(* CoDeSys 2.3.9.41 project: myLib.pro *)
(* Libraries: SysLibTime.lib 20.2.06 13:31:16, PID_Regulators.lib 28.12.06 17:47:54, Util.lib 18.5.10 15:14:28, STANDARD.LIB 4.10.05 11:14:46, IECSFC.LIB 13.4.06 15:51:28, ANALYZATION.LIB 5.10.99 09:05:06 *)

(* PLC configuration (modules and I/O channels)
Fast discrete inputs [I_SIMPLE_INPUT] node 0, in %IB0 out %QB0 {Filtrationtime = 10}
  DD1_DI0 AT %IX0.0 [BitInput] резерв
  DD1_DI1 AT %IX0.1 [BitInput] резерв
  DD1_DI2 AT %IX0.2 [BitInput] резерв
  DD1_DI3 AT %IX0.3 [BitInput] резерв
Discrete inputs [ID130] node 1, in %IB1 out %QB1 {Filtrationtime_GeneralINP = 10; Visibility = No; PinCount = 12}
  AT %IB1.0 [ByteInput] 8 discrete inputs
  AT %IB1.1 [ByteInput] 4 discrete inputs
Discrete outputs [ID131] node 2, in %IB2 out %QB2 {SafeValueByte = 0; SafeValueByteM = 0; Visibility = No; PinCount = 12}
  AT %QB2.0 [ByteOutput] 8 discrete outputs
  AT %QB2.1 [ByteOutput] 4 discrete outputs
Fast analog inputs [ID125] node 3, in %IB3 out %QB3 {Flt_Comm = 50Hz 2Por}
  DD1_AI0 AT %IR3.0 [FloatInputP] AI #1 - датчик температуры в помещении {AIN_TYPE = 4-20 mA; Peak_Filtr = 200; Flt_Ch = Off; TauRC = 10; MinFV = 0; MaxFV = 100}
  DD1_AI1 AT %IR3.1 [FloatInputP] AI #2 - расходомер FT01.01 (на входе, до отстойника) {AIN_TYPE = 4-20 mA; Peak_Filtr = 200; Flt_Ch = Off; TauRC = 10; MinFV = 0; MaxFV = 600}
  DD1_AI2 AT %IR3.2 [FloatInputP] AI #3 - расходомер FT01.02 (на выходе, после отстойника) {AIN_TYPE = 4-20 mA; Peak_Filtr = 200; Flt_Ch = Off; TauRC = 10; MinFV = 0; MaxFV = 600}
  DD1_AI3 AT %IR3.3 [FloatInputP] AI #4 - рН-метр QE01.01 (на входе, до отстойника) {AIN_TYPE = 4-20 mA; Peak_Filtr = 200; Flt_Ch = Off; TauRC = 10; MinFV = 0; MaxFV = 14}
  DD1_AI4 AT %IR3.4 [FloatInputP] AI #5 - рН-метр QE01.02 (на выходе, после отстойника) {AIN_TYPE = 4-20 mA; Peak_Filtr = 200; Flt_Ch = Off; TauRC = 10; MinFV = 0; MaxFV = 14}
  DD1_AI5 AT %IR3.5 [FloatInputP] AI #6 - сигнал от ФПК, давление на входе {AIN_TYPE = 4-20 mA; Peak_Filtr = 200; Flt_Ch = Off; TauRC = 10; MinFV = 0; MaxFV = 20000.0}
  DD1_AI6 AT %IR3.6 [FloatInputP] AI #7 - резерв {AIN_TYPE = 4-20 mA; Peak_Filtr = 200; Flt_Ch = Off; TauRC = 10; MinFV = 0; MaxFV = 20000.0}
  DD1_AI7 AT %IR3.7 [FloatInputP] AI #8 - обратная связь от ЧРП Н01.05 (частота, обороты, или ток) {AIN_TYPE = 4-20 mA; Peak_Filtr = 200; Flt_Ch = Off; TauRC = 10; MinFV = 0; MaxFV = 20000.0}
  AT %IW3.8 [WordInput] AI read time (10ms)
DD1_AO0 AT %QR4.0 [FloatOutputP] AO #1 - управление ЧРП Н01.05 (поддержание расхода по расходомеру FT01.02) {AOUT_TYPE = 4-20 mA; SafeValueREAL = 0.0}
DD1_AO1 AT %QR4.1 [FloatOutputP] AO #2 - управление ЧРП НД08.03/01 (подача флокулянта на входе, до отстойника, по FT01.01) {AOUT_TYPE = 4-20 mA; SafeValueREAL = 0.0}
DD1_AO2 AT %QR4.2 [FloatOutputP] AO #3 - управление ЧРП НД08.03/02 (подача флокулянта на входе, до отстойника, по FT01.01) {AOUT_TYPE = 4-20 mA; SafeValueREAL = 0.0}
DD1_AO3 AT %QR4.3 [FloatOutputP] AO #4 - управление НД05.02/01 (подача 10%NaCl из УПГ на входе, до отстойника, по FT01.01) {AOUT_TYPE = 4-20 mA; SafeValueREAL = 0.0}
Special input [ID103] node 5, in %IB5 out %QB5 {Filtrationtime = 1000; PinCount = 1; WatchDogPeriod = 400; PollPeriod = 3000; Visibility = No}
  AT %IX5.0 [BitInput] Special input
Special output [ID104] node 6, in %IB6 out %QB6 {Visibility = No; PinCount = 1}
  AT %QX6.0 [BitOutput] Special output
ModBus (Master) [MODBUS_MASTER_ID450] node 7, in %IB7 out %QB7 {Visibility = No}
  AT %QD7.0 [DWordOutput] Last address
  AT %QW7.1 [WordOutput] Last error
  RS-485-1 [COM1_USART] node 0, in %IB7.0 out %QB7.0 {CommunicationSpeed = 57600; Parity = NO PARITY CHECK; BitLength = 8 bits; StopLength = One stop bit; InterfaceType = RS485; FrameOriented = RTU; Timeout = 0; Visibility = No}
  Universal Modbus device [ID2000] node 1, in %IB7.1 out %QB7.1 {ModuleIP = 10:0:0:102; ServiceTimeout = 20; TCPport = 502; NetMode = Serial; ModuleSlaveAddress = 2; RequestType = Both; PeriodOfService = 100; Visibility = No; RepeatCounter = 0; ByteSequence = Trace_mode}
    AT %QB7.1.0 [ComChannel] Command (0xff - Start)
DD2_DO AT %QD7.1.0.0 [DWordOutput] регистр 0, команда 0х0f
Universal Modbus device [ID2000] node 2, in %IB7.2 out %QB7.2 {ModuleIP = 10:0:0:103; ServiceTimeout = 20; TCPport = 502; NetMode = Serial; ModuleSlaveAddress = 3; RequestType = Both; PeriodOfService = 100; Visibility = No; RepeatCounter = 0; ByteSequence = Trace_mode}
  AT %QB7.2.0 [ComChannel] Command (0xff - Start)
DD3_DO AT %QD7.2.0.0 [DWordOutput]
Universal Modbus device [ID2000] node 3, in %IB7.3 out %QB7.3 {ModuleIP = 10:0:0:104; ServiceTimeout = 20; TCPport = 502; NetMode = Serial; ModuleSlaveAddress = 4; RequestType = Both; PeriodOfService = 100; Visibility = No; RepeatCounter = 0; ByteSequence = Trace_mode}
  AT %QB7.3.0 [ComChannel] Command (0xff - Start)
  32bit output module [ID2006] node 0, in %IB7.3.0 out %QB7.3.0 {ModbusAddress = 0; Command_write_regs = Force multiple coils (0x0f); Visibility = No}
    DD4_DO AT %QD7.3.0.0 [DWordOutput]
Universal Modbus device [ID2000] node 4, in %IB7.4 out %QB7.4 {ModuleIP = 10:0:0:105; ServiceTimeout = 20; TCPport = 502; NetMode = Serial; ModuleSlaveAddress = 5; RequestType = Both; PeriodOfService = 100; Visibility = No; RepeatCounter = 0; ByteSequence = Trace_mode}
  AT %QB7.4.0 [ComChannel] Command (0xff - Start)
DD5_DI AT %ID7.4.0.0 [DWordInput]
Universal Modbus device [ID2000] node 5, in %IB7.5 out %QB7.5 {ModuleIP = 10:0:0:106; ServiceTimeout = 20; TCPport = 502; NetMode = Serial; ModuleSlaveAddress = 6; RequestType = Both; PeriodOfService = 100; Visibility = No; RepeatCounter = 0; ByteSequence = Trace_mode}
  AT %QB7.5.0 [ComChannel] Command (0xff - Start)
DD6_DI AT %ID7.5.0.0 [DWordInput]
Universal Modbus device [ID2000] node 6, in %IB7.6 out %QB7.6 {ModuleIP = 10:0:0:107; ServiceTimeout = 20; TCPport = 502; NetMode = Serial; ModuleSlaveAddress = 7; RequestType = Both; PeriodOfService = 100; Visibility = No; RepeatCounter = 0; ByteSequence = Trace_mode}
  AT %QB7.6.0 [ComChannel] Command (0xff - Start)
DD7_DI AT %ID7.6.0.0 [DWordInput]
Universal Modbus device [ID2000] node 7, in %IB7.7 out %QB7.7 {ModuleIP = 10:0:0:108; ServiceTimeout = 20; TCPport = 502; NetMode = Serial; ModuleSlaveAddress = 8; RequestType = Both; PeriodOfService = 100; Visibility = No; RepeatCounter = 0; ByteSequence = Trace_mode}
  AT %QB7.7.0 [ComChannel] Command (0xff - Start)
DD8_DI AT %ID7.7.0.0 [DWordInput]
Universal Modbus device [ID2000] node 8, in %IB7.8 out %QB7.8 {ModuleIP = 10:0:0:109; ServiceTimeout = 20; TCPport = 502; NetMode = Serial; ModuleSlaveAddress = 9; RequestType = Both; PeriodOfService = 100; Visibility = No; RepeatCounter = 0; ByteSequence = Trace_mode}
  AT %QB7.8.0 [ComChannel] Command (0xff - Start)
DD9_DI AT %ID7.8.0.0 [DWordInput]
AT %QB7.9.0 [ComChannel] Command (0xff - Start)
DD10_AO0 AT %QW7.9.0.0 [WordOutput] управление 4...20мА НД05.02/01
DD10_AO1 AT %QW7.9.1.0 [WordOutput]
DD10_AO2 AT %QW7.9.2.0 [WordOutput]
DD10_AO3 AT %QW7.9.3.0 [WordOutput]
DD10_AO4 AT %QW7.9.4.0 [WordOutput]
DD10_AO5 AT %QW7.9.5.0 [WordOutput]
DD10_AO6 AT %QW7.9.6.0 [WordOutput]
DD10_AO7 AT %QW7.9.7.0 [WordOutput]
*)

(* Global variable list: Global_Variables *)
VAR_GLOBAL
	wordMaxValue: WORD := 65535;		(*max value of WORD.*)
END_VAR

(* POU PLC_PRG, CFC *)
PROGRAM PLC_PRG
VAR
	temperatureLimits: LIMITALARM;		(*блок контроля границ допустимой температуры в помещении*)
	alarmHighTemperature: BOOL;		(*температура выше заданного диапазона*)
	alarmLowTemperature: BOOL;		(*температура ниже заданного диапазона*)
	temperatureValue: REAL;		(*значение температуры в помещении*)
	DD1_AI0_temperature: DECODE_FLOAT;		(*блок контроля состояния аналогового входа ПЛК для датчика температуры в помещении*)
	DD1_AI1_flow: DECODE_FLOAT;		(*блок контроля состояния аналогового входа ПЛК для расходомера FT01.01*)

	ND0502dosing: DosingPumpProportional;		(*Блок управления дозированием насосов НД05.02/01 и НД05.02/02.
			Пропорционально расходу по FT01.01*)
	ND0502regime: choosePumpRegime;		(*Блок выбора режима включения НД05.02/01 и НД05.02/02.*)
	ND0502manager: TwoPumpManager;		(*Блок управления включением дозирующих насосов
			НД05.02/01 и НД05.02/02.*)

	ND0602dosing: DosingPumpProportional;		(*Блок управления дозированием насосов НД06.02/01 и НД06.02/02.
			Пропорционально расходу по FT01.02.*)
	ND0602regime: choosePumpRegime;		(*Блок выбора режима включения НД06.02/01 и НД06.02/02.*)
	ND0602manager: TwoPumpManager;		(*Блок управления включением дозирующих насосов
			НД06.02/01 и НД06.02/02.*)

	ND0603dosing: DosingPumpProportional;		(*Блок управления дозированием насосов НД06.03/01 и НД06.03/02.
						Пропорционально расходу по FT01.01*)
	ND0603regime: choosePumpRegime;		(*Блок выбора режима включения НД06.03/01 и НД06.03/02.*)
	ND0603manager: TwoPumpManager;		(*Блок управления включением дозирующих насосов
						НД06.03/01 и НД06.03/02.*)

	ND0703pidReg: PID;		(*Блок автоматического поддержания заданного значения рН стоков подачей щелочи через НД07.03
								по показаниям QE01.01.*)
	ND0703regime: choosePumpRegime;		(*Блок выбора режима включения НД07.03/01 и НД07.03/02.*)
	ND0703manager: TwoPumpManager;		(*Блок управления включением дозирующих насосов
									НД07.03/01 и НД07.03/02*)

	ND0803dosing: DosingPumpProportional;		(*Блок управления дозированием насосов НД08.03*)
	ND0803regime: choosePumpRegime;		(*Блок выбора режима включения насосов НД08.03.*)
	ND0803manager: TwoPumpManager;		(*Блок управления включением дозирующих насосов НД08.03.*)

	ND0804linearTransformator: LIN_TRAFO;		(*Блок преобразования сигнала на управление от 0 до 100% в 4...20мА*)

	DD1_AI1_FT0101: DECODE_FLOAT;		(*Блок контроля аналогового входа DD1_AI1 (расходомер FT01.01)*)
	DD1_AI2_FT0102: DECODE_FLOAT;		(*блок контроля состояния аналогового входа ПЛК для расходомера FT01.02*)
	DD1_AI3_QE0101: DECODE_FLOAT;		(*блок контроля состояния аналогового входа ПЛК для рН-метра QE01.01*)
	DD1_AI4_QE0102: DECODE_FLOAT;		(*блок контроля состояния аналогового входа ПЛК для рН-метра QE01.02*)

	DD1_AI1_FT0101value: REAL;		(*Показания расходомера FT01.01 после блока контроля аналогового входа ПЛК.*)
	DD1_AI2_FT0102value: REAL;		(*Показания расходомера FT01.02 после блока контроля аналогового входа ПЛК.*)
	DD1_AI3_QE0101value: REAL;		(*Показания рН-метра QE01.01 после блока контроля аналогового входа ПЛК.*)
	DD1_AI4_QE0102value: REAL;		(*Показания рН-метра QE01.02 после блока контроля аналогового входа ПЛК*)

	N0105manager: TwoPumpManager;		(*Блок управления включением насосов Н01.05*)
	N0105regime: choosePumpRegime;		(*Блок выбора режима включения Н05.01*)
	N0105pidReg: PID;		(*Блок автоматического поддержания заданного значения расхода по показаниям FT01.02*)
	N0105regByC: RS;		(*Триггер выбора режима по количеству включений.*)
	N0105regByWT: RS;		(*Триггер выбора режима по наработке.*)
	N0105managerKM1off: BOOL;		(*Переменная управления состоянием контактора питания ЧРП (КМ1).*)
	N0105rsTrigKM1: RS;		(*Триггер управления состоянием контактора КМ1. Постоянно включен.
			Выключается если N0105managerKM1off=true.*)
	N0105timerKM1off: TOF;		(*Таймер отключения КМ1. Срабатывает по импульсу на входе.
			Выключается через заданное в N0105switchKM1Delay время.*)
	N0105switchKM1Delay: TIME := T#20S;		(*Время отключения питания ЧРП Н01.05.
			По умолчанию = 20 сек.*)
	N010501rTrig: R_TRIG;		(*Детектор перенего фронта сигнала выбора режима Н01.05/01 = главный.*)
	N010501fTrig: F_TRIG;		(*Детектор спада сигнала выбора режима Н01.05/01 = главный.*)
	N0105trigKM2on: RS;		(*Триггер включения КМ2.*)
	N0105switchKM2Delay: TON;		(*Таймер задержки включения КМ2.*)
	N0105switchKM23Delay: TIME := T#15s;		(*Время задержки включения КМ2 и КМ3 при переключении.
			По умолчанию 15 сек.*)
	N010502rTrig: R_TRIG;		(*Детектор перенего фронта сигнала выбора режима Н01.05/02 = главный.*)
	N010502fTrig: F_TRIG;		(*Детектор спада сигнала выбора режима Н01.05/02 = главный.*)
	N0105trigKM3on: RS;		(*Триггер включения КМ3.*)
	N0105switchKM3Delay: TON;		(*Таймер задержки включения КМ3.*)

	rTrigStartInitializer: R_TRIG;		(*Детектор переднего фронта,
			инициализирует булевы переменные при старте программы.*)
	startInitializer: BOOL;		(*Инициализирует булевы переменные при старте программы.*)

	N0105sttartTrig: RS;		(*Триггер запуска насосов Н01.05 по датчикам уровня.*)

	N010501alarm: BOOL;		(*Авария насоса Н01.05/01*)
	N010502alarm: BOOL;		(*Авария насоса Н01.05/02*)
	N010501toStart: BOOL;		(*Промежуточный сигнал о необходимости запуска Н01.05/01.*)
	N010502toStart: BOOL;		(*Промежуточный сигнал о необходимости запуска Н01.05/02.*)
	N0105minFlow: REAL := 10;		(*Минимальное значение расхода для подачи сигнала на начало дозирования.
			По умолчанию, если ничего не подключено ко входу, равно 10 кубометров в час.*)
	N0105f_trigStop: F_TRIG;		(*Детектор останова насоса кнопкой со щита (спад сигнала включенного реле).*)
	N010501alarmTrig: RS;		(*Триггер аварии насоса Н01.05/01.*)
	N010502alarmTrig: RS;		(*Триггер аварии насоса Н01.05/02.*)



	tempN0105switchKM1off: BOOL;		(*temporary variable to switch off KM1 when pumps change.*)
	tempN010501Trig: RS;		(*temporary trigger to catch N010501 start impuls.*)
	tempN010502Trig: RS;		(*temporary trigger to catch N01.05/02 start impuls*)
	tempN0105rTrigKM1off: R_TRIG;		(*temporary rising front detector to switch off KM1 = drive power supply.*)
	tempN010501rTrig: R_TRIG;		(*temporary rising signal to start N010501 detector*)
	tempN010502rTrig: R_TRIG;		(*temporary rising signal to start N010502 detector*)
	tempN0105RMswitchDelay: BOOL;		(*Init temporaty delay to switch KM2 or KM3.*)
	tempN0105delayOUT: BOOL;		(*temporari signal that delay to switch is over.*)
	tempN0105switchKM2offDelay: TOF;		(*temporary delay to switch off KM2*)
	tempN0105switchKM3offDelay: TOF;		(*temporary delay to switch off KM3*)
	tempN0105switchKMoffDelay: TIME := T#3s;		(*temporary switch off RM delay.*)
	tempN0105ready: BOOL;		(*Temporary variable shows that system is ready to start pump.*)
	tempN0105readyToStart: TON;		(*Temporary ready to start delay timer.*)
	tempN0105readyToStartDelay: TIME := T#5s;		(*temporary delay to show signal that system is ready to start.
			Init value = 5sec.*)
	tempTwoPumpOneDriveManager: TwoPumpOneDriveManager;		(*test*)
	temp1: BOOL;
	temp2: BOOL;
	temp3: BOOL;
	temp4: BOOL;
	temp5: BOOL;
	temp6: BOOL;
	temp7: BOOL;
	temp8: BOOL;
	temp9: BOOL;
	temp10: BOOL;
	temp11: BOOL;
	temp12: WORD;
	temp13: WORD;
	temp14: TIME;
	temp15: TIME;
	temp16: BOOL;
	temp17: BOOL;
	temp18: BOOL;
	temp19: BOOL;
END_VAR
VAR_INPUT
	alarmReset: BOOL;		(*Сброс аварий.*)

	ND0502resetCountP1: BOOL;		(*Сбросить счетчик количества включений НД05.02/01.*)
	ND0502resetCountP2: BOOL;		(*Сбросить счетчик количества включений НД05.02/02.*)
	ND0502resetWorkTimeP1: BOOL;		(*Сбросить счетчик наработки НД05.02/01.*)
	ND0502resetWorkTimeP2: BOOL;		(*Сбросить счетчик наработки НД05.02/02.*)

	ND0602resetCountP1: BOOL;		(*Сбросить счетчик количества включений НД06.02/01.*)
	ND0602resetCountP2: BOOL;		(*Сбросить счетчик количества включений НД06.02/02.*)
	ND0602resetWorkTimeP1: BOOL;		(*Сбросить счетчик количества наработки НД06.02/01.*)
	ND0602resetWorkTimeP2: BOOL;		(*Сбросить счетчик количества наработки НД06.02/02.*)

	ND0603resetCountP1: BOOL;		(*Сбросить счетчик количества включений НД06.03/01.*)
	ND0603resetCountP2: BOOL;		(*Сбросить счетчик количества включений НД06.03/02.*)
	ND0603resetWorkTimeP1: BOOL;		(*Сбросить счетчик времени наработки НД06.03/01.*)
	ND0603resetWorkTimeP2: BOOL;		(*Сбросить счетчик времени наработки НД06.03/02.*)

	ND0703resetCountP1: BOOL;		(*Сбросить счетчик количества включений НД07.03/01.*)
	ND0703resetCountP2: BOOL;		(*Сбросить счетчик количества включений НД07.03/02.*)
	ND0703resetWorkTimeP1: BOOL;		(*Сбросить счетчик наработки НД07.03/01.*)
	ND0703resetWorkTimeP2: BOOL;		(*Сбросить счетчик наработки НД07.03/02.*)
	ND0703YoutManual: REAL;		(*Задание значения выходу Y в ручном режиме (4...20мА).*)
	ND0703YmanAuto: BOOL;		(*Выбор управления выходом Y в ручном или автоматическом режиме.*)

	ND0803resetCountP1: BOOL;		(*Сброс счетчика количества включений НД08.03/01.*)
	ND0803resetCountP2: BOOL;		(*Сброс счетчика количества включений НД08.03/02.*)
	ND0803resetWorkTimeP1: BOOL;		(*Сброс счетчика наработки НД08.03/01.*)
	ND0803resetWorkTimeP2: BOOL;		(*Сброс счетчика наработки НД08.03/02.*)

	N0105YoutManual: REAL;		(*Задание значения выходу Y в ручном режиме (4...20мА).*)
	N0105YmanAuto: BOOL;		(*Выбор управления выходом Y в ручном или автоматическом режиме.*)

END_VAR
VAR_OUTPUT
	ND0502dosingError: BOOL;		(*Ошибка дозирования НД05.02.
			Проверить заданные уставки.*)
	ND0502statRegimeP1M: BOOL;		(*статус: режим НД05.02 - насос 1 = главный.*)
	ND0502statRegimeP2M: BOOL;		(*статус: режим НД05.02 - насос 2 = главный*)
	ND0502statRegimeByC: BOOL;		(*статус: режим НД05.02 - по количеству включений*)
	ND0502statRegimeByWT: BOOL;		(*статус: режим НД05.02 - по наработке*)

	ND0602dosingError: BOOL;		(*Ошибка дозирования НД06.02/01-02.
						Проверить заданные уставки.*)
	ND0602statRegimeP1M: BOOL;		(*статус: режим НД0602 - насос 1 = главный.*)
	ND0602statRegimeP2M: BOOL;		(*статус: режим НД06.02 - насос 2 = главный.*)
	ND0602statRegimeByC: BOOL;		(*статус: режим НД06.02 - по количеству включений.*)
	ND0602statRegimeByWT: BOOL;		(*статус: режим НД06.02 - по наработке.*)

	ND0603dosingError: BOOL;		(*Ошибка дозирования НД06.03.
						Проверить заданные уставки.*)
	ND0603statRegimeP1M: BOOL;		(*статус: режим НД0603 - насос 1 = главный.*)
	ND0603statRegimeP2M: BOOL;		(*статус: режим НД0603 - насос 2 = главный.*)
	ND0603statRegimeByC: BOOL;		(*статус: режим НД06.03 - по количеству включений.*)
	ND0603statRegimeByWT: BOOL;		(*статус: режим НД06.03 - по наработке.*)

	ND0703statRegimeP1M: BOOL;		(*статус: режим НД0703 - насос 1 = главный.*)
	ND0703statRegimeP2M: BOOL;		(*статус: режим НД0703 - насос 2 = главный.*)
	ND0703statRegimeByC: BOOL;		(*статус: режим НД07.03 - по количеству включений.*)
	ND0703statRegimeByWT: BOOL;		(*статус: режим НД07.03 - по наработке.*)

	ND0803dosingError: BOOL;		(*Ошибка блока дозирования НД08.03.*)
	ND0803statRegimeP1M: BOOL;		(*статус: режим НД08.03 - насос 1 = главный*)
	ND0803statRegimeP2M: BOOL;		(*статус: режим НД08.03 - насос 2 = главный*)
	ND0803statRegimeByC: BOOL;		(*статус: режим НД08.03 - по количеству включений*)
	ND0803statRegimeByWT: BOOL;		(*статус: режим НД08.03 - по наработке.*)

	ND0804dosingError: BOOL;		(*Ошибка дозирования НД08.04. Проверь уставки.*)

	DD1_AI0_error: BOOL;		(*авария входа AI1 (возможно, обрыв)*)
	DD1_AI1_error: BOOL;		(*авария входа AI2 (возможно, обрыв)*)
	DD1_AI2_error: BOOL;		(*авария входа AI3 (возможно, обрыв)*)
	DD1_AI3_error: BOOL;		(*авария входа AI4 (возможно, обрыв)*)
	DD1_AI4_error: BOOL;		(*авария входа AI5 (возможно, обрыв)*)

	N0105statRegimeP1M: BOOL;		(*статус: режим Н01.05/01 = главный.*)
	N0105statRegimeP2M: BOOL;		(*статус: режим Н01.05/02 = главный.*)
	N0105statRegimeByC: BOOL;		(*статус: режим Н01.05 = по количеству включений.*)
	N0105statRegimeByWT: BOOL;		(*статус: режим Н01.05 = по наработке.*)

END_VAR
VAR RETAIN
	maxTemperature: BYTE;		(*Температура, выше которой будет подан сигнал ВЫСОКАЯ ТЕМПЕРАТУРА*)
	minTemperature: BYTE;		(*температура, ниже которой будет подан сигнал НИЗКАЯ ТЕМПЕРАТУРА*)

END_VAR
VAR_INPUT RETAIN
	ND0502setMaxDosVal: REAL;		(*Указать максимальную производительность НД05.02.*)
	ND0502setKoefProp: REAL;		(*Задать количество реагента в мл на один кубометр стоков.*)
	ND0502regimeP1M: BOOL := 1;		(*Выбор режима включения доз.насосов НД05.02: первый насос - главный.
			Выбрано по умолчанию до выбора пользователя.*)
	ND0502regimeP2M: BOOL;		(*Выбор режима включения доз.насосов НД05.02:
			второй насос - главный.*)
	ND0502regimeByWT: BOOL;		(*Выбор режима включения доз.насосов НД05.02:
			по наработке.*)
	ND0502regimeByC: BOOL;		(*Выбор режима включения доз.насосов НД05.02:
			по количеству включений.*)

	ND0602setMaxDosVal: REAL;		(*Указать максимальную производительность НД06.02.*)
	ND0602setKoefProp: REAL;		(*Задать количество реагента в мл на один кубометр стоков.*)
	ND0602regimeP1M: BOOL := 1;		(*Выбор режима включения доз.насосов НД06.02: первый насос - главный.
			Выбрано по умолчанию до выбора пользователя.*)
	ND0602regimeP2M: BOOL;		(*Выбор режима включения доз.насосов НД06.02: второй насос - главный.
			*)
	ND0602regimeByWT: BOOL;		(*Выбор режима включения доз.насосов НД06.02:
			по наработке.*)
	ND0602regimeByC: BOOL;		(*Выбор режима включения доз.насосов НД06.02:
			по количеству включений.*)

	ND0603setMaxDosVal: REAL;		(*Указать максимальную производительность НД06.03.*)
	ND0603setKoefProp: REAL;		(*Задать количество реагента в мл на один кубометр стоков.*)
	ND0603regimeP1M: BOOL := 1;		(*Выбор режима включения доз.насосов НД06.03: первый насос - главный.
			Выбрано по умолчанию до выбора пользователя.*)
	ND0603regimeP2M: BOOL;		(*Выбор режима включения доз.насосов НД06.03: второй насос - главный.*)
	ND0603regimeByWT: BOOL;		(*Выбор режима включения доз.насосов НД06.03:
			по наработке.*)
	ND0603regimeByC: BOOL;		(*Выбор режима включения доз.насосов НД06.03:
			по количеству включений.*)

	ND0703pHsetValue: REAL := 7.5;		(*Задание рН для поддержания подачей щелочи НД07.03 и контроля по QE01.01.*)
	ND0703regimeP1M: BOOL := 1;		(*Выбор режима включения доз.насосов НД07.03: первый насос - главный.
						Выбрано по умолчанию до выбора пользователя.*)
	ND0703regimeP2M: BOOL;		(*Выбор режима включения доз.насосов НД07.03: второй насос - главный*)
	ND0703regimeByWT: BOOL;		(*Выбор режима включения доз.насосов НД07.03: по наработке.*)
	ND0703regimeByC: BOOL;		(*Выбор режима включения доз.насосов НД07.03: по количеству включений.*)
	ND0703koeffI: REAL := 10;		(*Коэффициент интегральной части ПИД. По умолчанию = 10.*)
	ND0703koeffD: REAL := 1;		(*Коэффициент дифференциальной части ПИД. По умолчанию = 1.*)
	ND0703koeffP: REAL := 1;		(*Коэффициент пропорциональной части ПИД. По умолчанию = 1.*)

	ND0803setMaxDosVal: REAL;		(*Указать максимальную производительность НД08.03*)
	ND0803setKoefProp: REAL;		(*Задать количество реагента в мл на один кубометр стоков.*)
	ND0803regimeP1M: BOOL := 1;		(*Выбор режима включения доз.насосов НД08.03: первый насос - главный.
									Выбрано по умолчанию до выбора пользователя.*)
	ND0803regimeP2M: BOOL;		(*Выбор режима включения доз.насосов НД08.03: второй насос - главный.*)
	ND0803regimeByWT: BOOL;		(*Выбор режима включения доз.насосов НД08.03: по наработке.*)
	ND0803regimeByC: BOOL;		(*Выбор режима включения доз.насосов НД08.03: по количеству включений.*)

	ND0804doseValue: BYTE;		(*Задание на дозирование НД0804 в процентах от максимальной производительности (0-100).*)

	N0105regimeByC: BOOL;		(*Выбор режима запуска Н01.05: по количеству включений.
			*)
	N0105regimeByWT: BOOL;		(*Выбор режима запуска Н01.05: по наработке.*)
	N0105flowSetValue: REAL := 72;		(*Задание расхода для поддержания ЧРП Н01.05 по расходомеру FT01.02.
			По умолчанию = 72 кубометра в час.*)
	N0105koeffP: REAL := 1;		(*Коэффициент пропорциональной части ПИД. По умолчанию = 1.*)
	N0105koeffI: REAL := 10;		(*Коэффициент интегральной части ПИД. По умолчанию = 10.*)
	N0105koeffD: REAL := 1;		(*Коэффициент дифференциальной части ПИД. По умолчанию = 1.*)

END_VAR
VAR_OUTPUT RETAIN
	ND0502counterP1: WORD;		(*Счетчик количества включений НД05.02/01.*)
	ND0502counterP2: WORD;		(*Счетчик количества включений НД05.02/02.*)
	ND0502workTimeP1: TIME;		(*Счетчик времени наработки НД05.02/01.*)
	ND0502workTimeP2: TIME;		(*Счетчик времени наработки НД05.02/02.*)

	ND0602counterP1: WORD;		(*Счетчик количества включений НД06.02/01.*)
	ND0602counterP2: WORD;		(*Счетчик количества включений НД06.02/02.*)
	ND0602workTimeP1: TIME;		(*Счетчик времени наработки НД06.02/01.*)
	ND0602workTimeP2: TIME;		(*Счетчик времени наработки НД06.02/02.*)

	ND0603counterP1: WORD;		(*Счетчик количества включений НД06.03/01.*)
	ND0603counterP2: WORD;		(*Счетчик количества включений НД06.03/02.*)
	ND0603workTimeP1: TIME;		(*Счетчик времени наработки НД06.03/01.*)
	ND0603workTimeP2: TIME;		(*Счетчик времени наработки НД06.03/02.*)

	ND0703counterP1: WORD;		(*Счетчик количества включений НД07.03/01.*)
	ND0703counterP2: WORD;		(*Счетчик количества включений НД07.03/02.*)
	ND0703workTimeP1: TIME;		(*Счетчик времени наработки НД07.03/01.*)
	ND0703workTimeP2: TIME;		(*Счетчик времени наработки НД07.03/02.*)

	ND0803counterP1: WORD;		(*Счетчик количества включений НД08.03/01.*)
	ND0803counterP2: WORD;		(*Счетчик количества включений НД08.03/02.*)
	ND0803workTimeP1: TIME;		(*Счетчик времени наработки НД08.03/01.*)
	ND0803workTimeP2: TIME;		(*Счетчик времени наработки НД08.03/02.*)

	N0105counterP1: WORD;		(*Счетчик количества включений Н01.05/01.*)
	N0105counterP2: WORD;		(*Счетчик количества включений Н01.05/02.*)
	N0105workTimeP1: TIME;		(*Счетчик времени наработки Н01.05/01.*)
	N0105workTimeP2: TIME;		(*Счетчик времени наработки Н01.05/02.*)
END_VAR
VAR (* helpers for the ST form of the networks *)
	_t977 : WORD;
	_t899 : WORD;
	_t831 : REAL;
	_t801 : WORD;
	_t1027 : WORD;
	_t1033 : WORD;
	_t1355 : REAL;
	_t1361 : REAL;
	_t1183 : WORD;
	_t1189 : WORD;
	_t1404 : BOOL;
	_t1403 : BOOL;
END_VAR
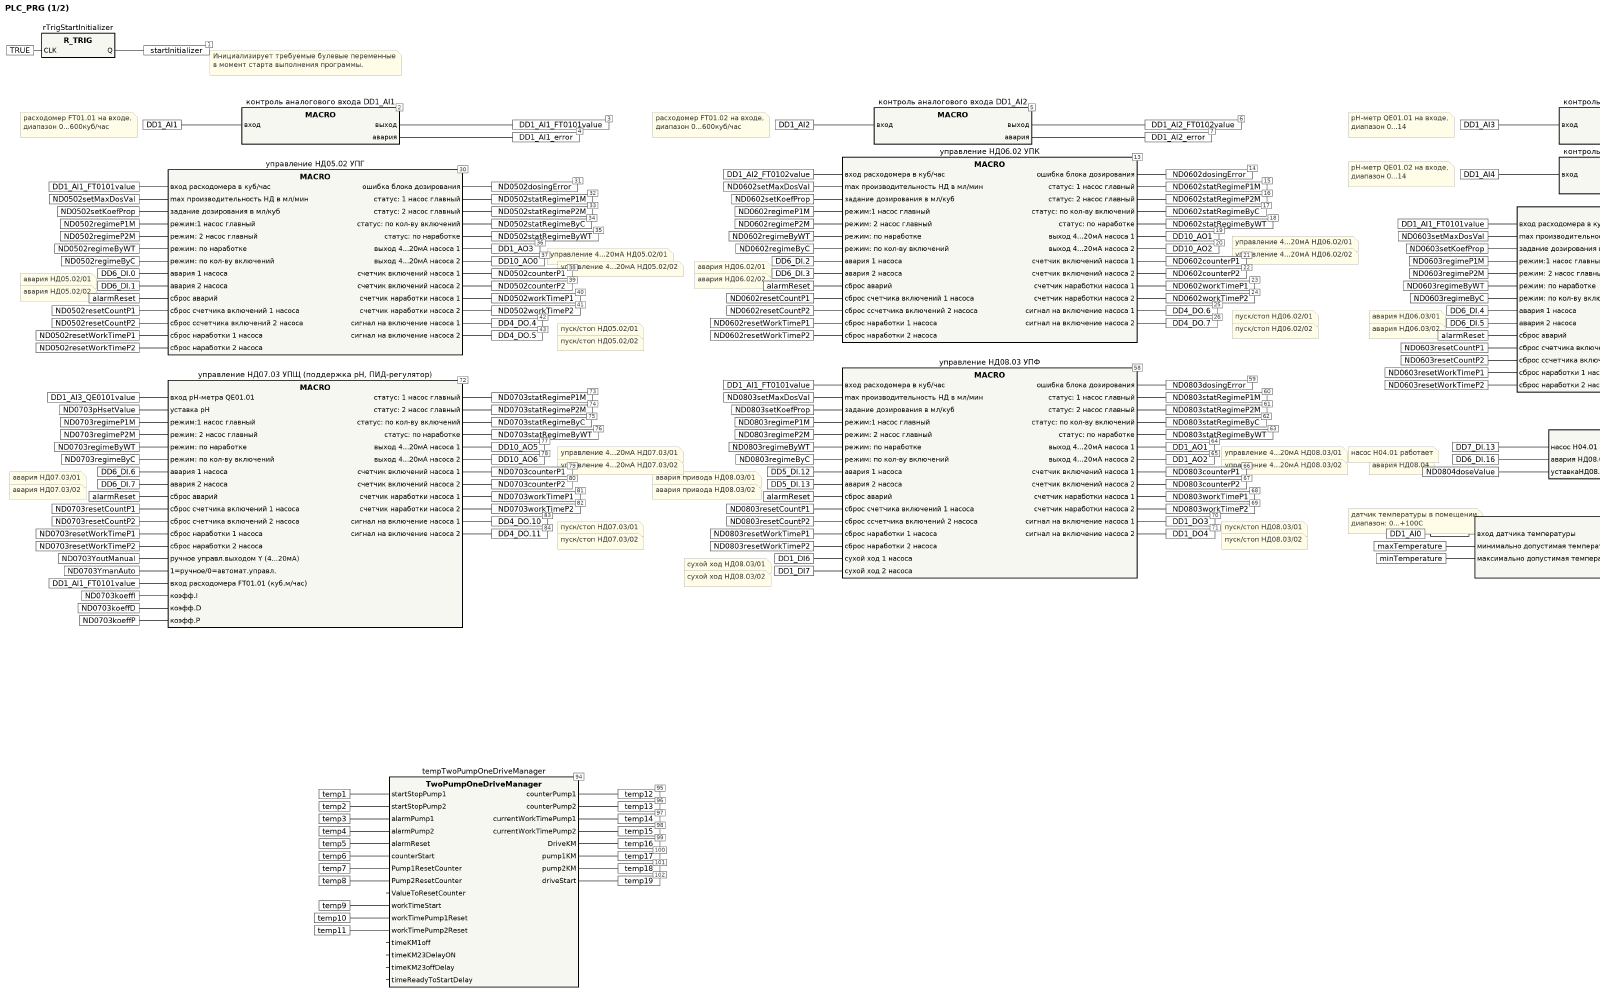
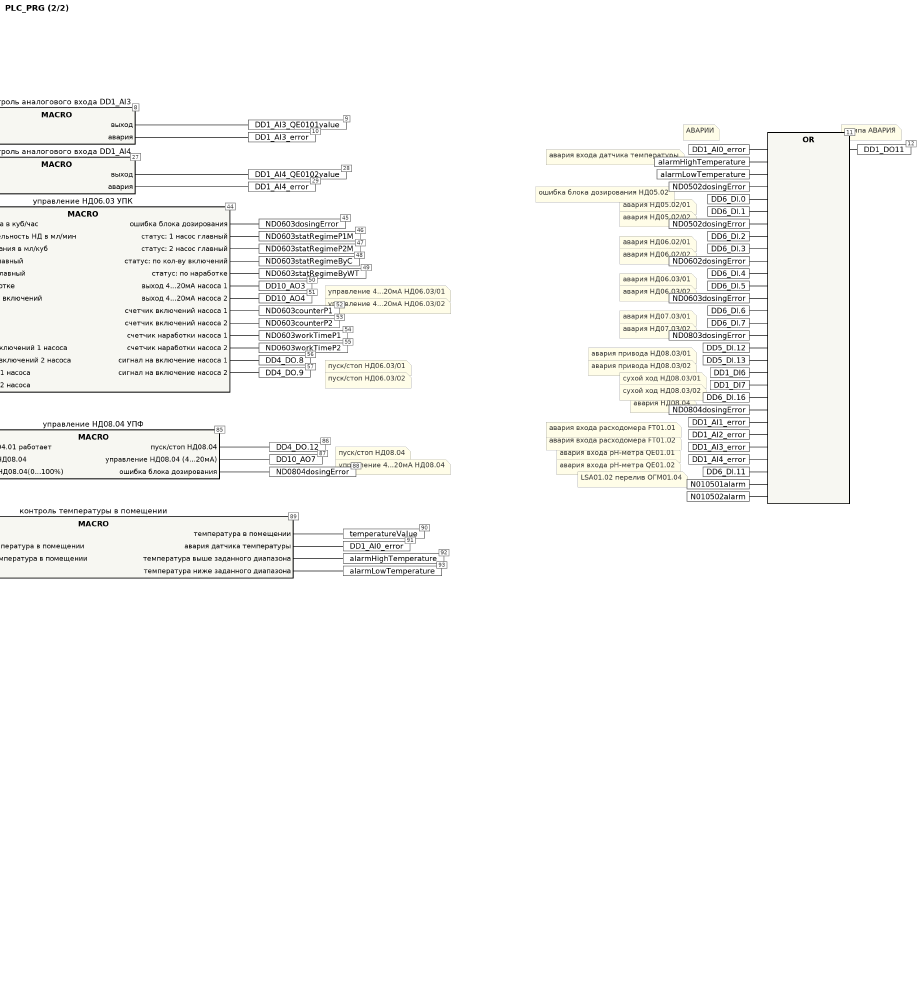
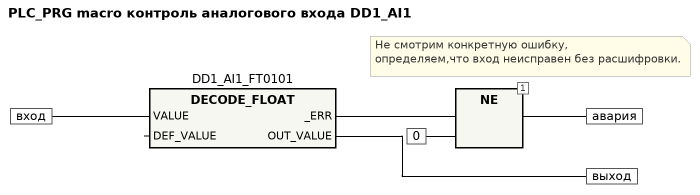
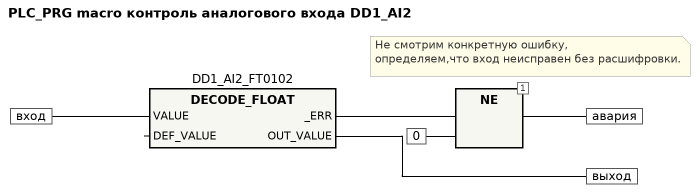
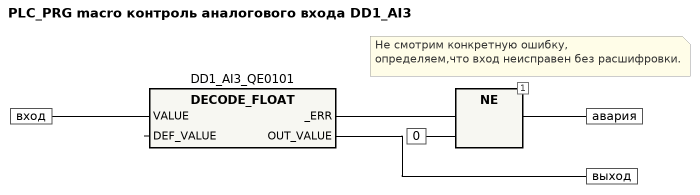
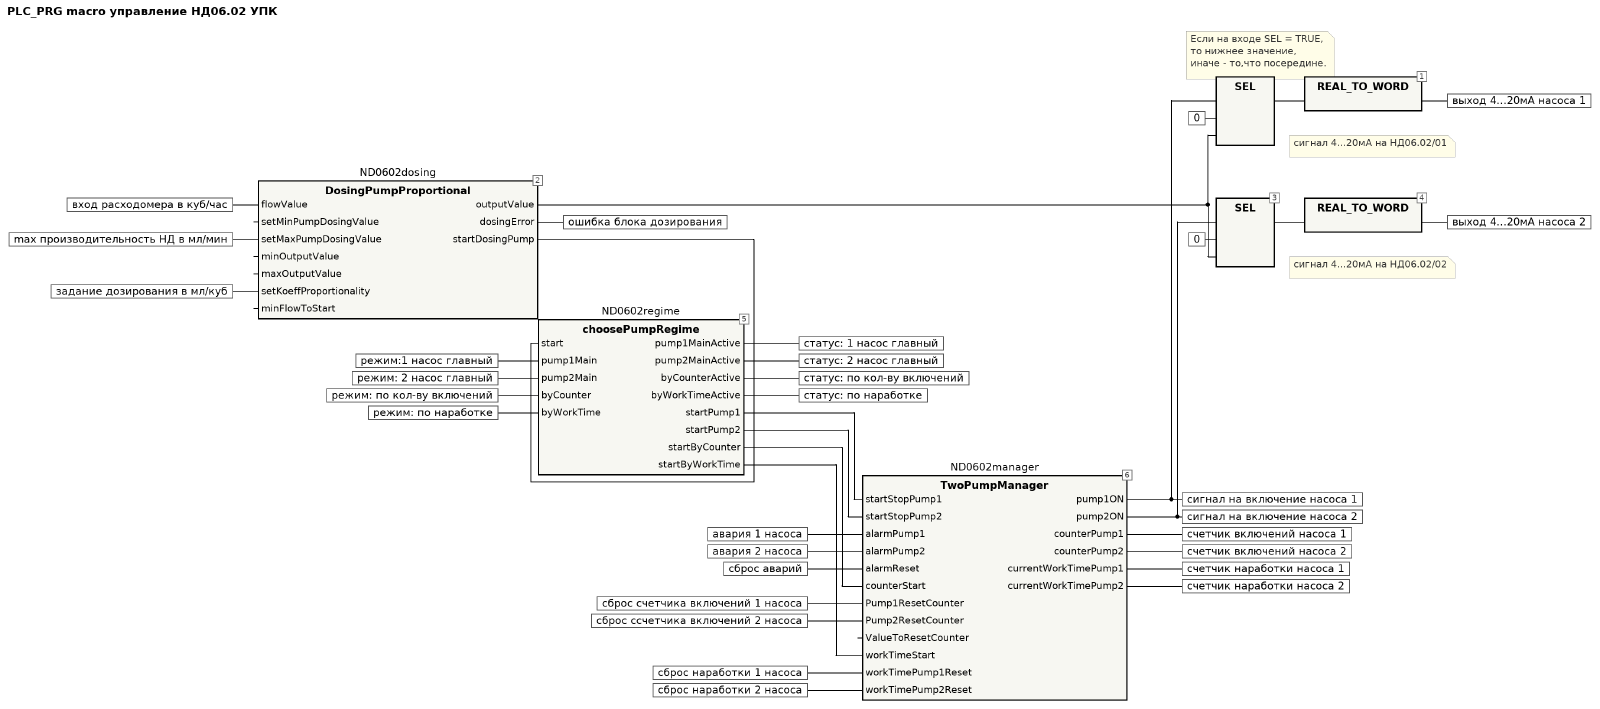
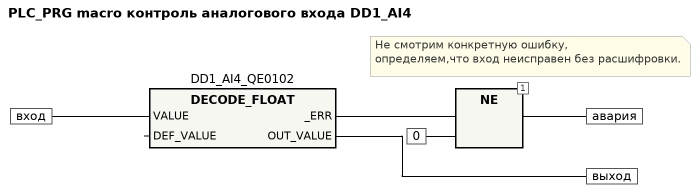
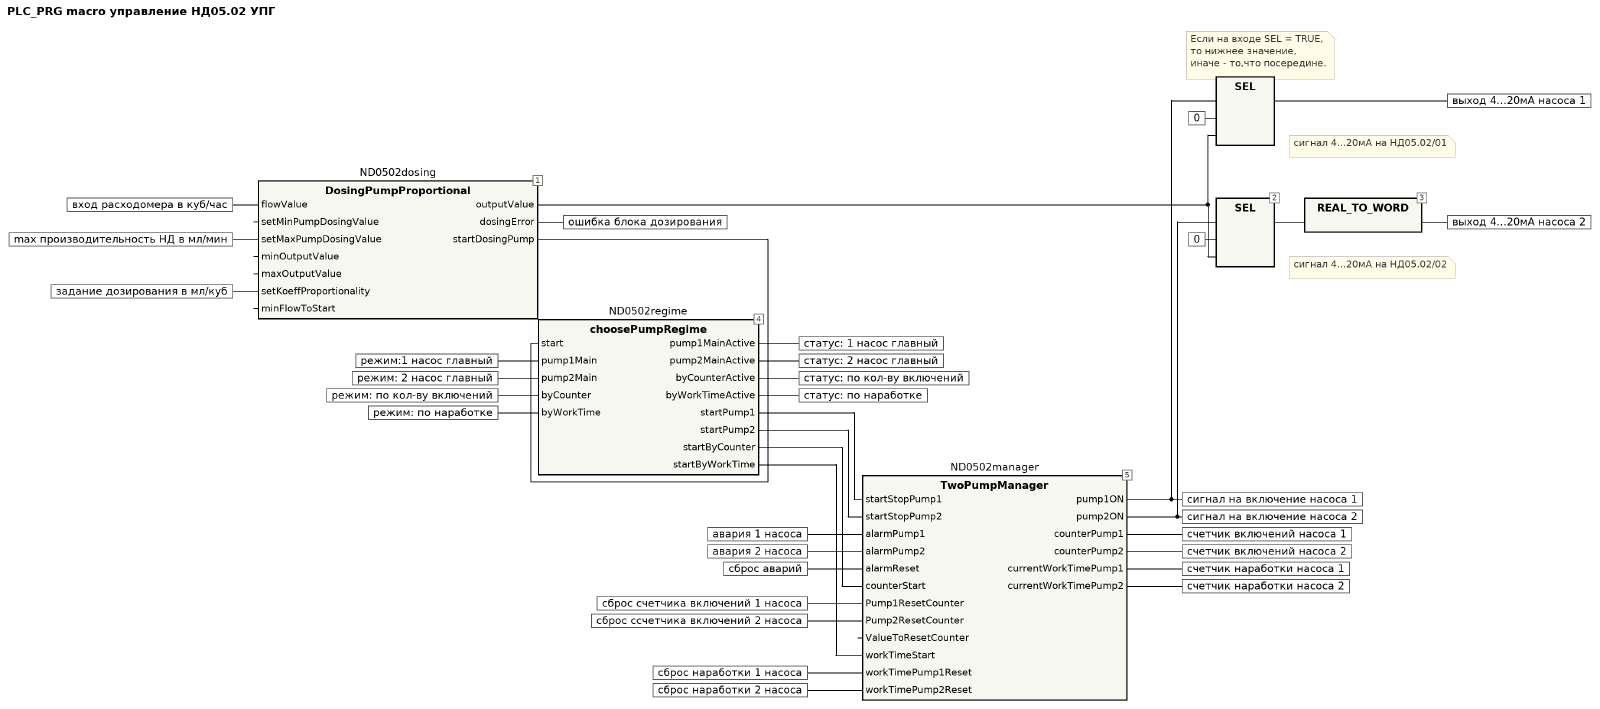
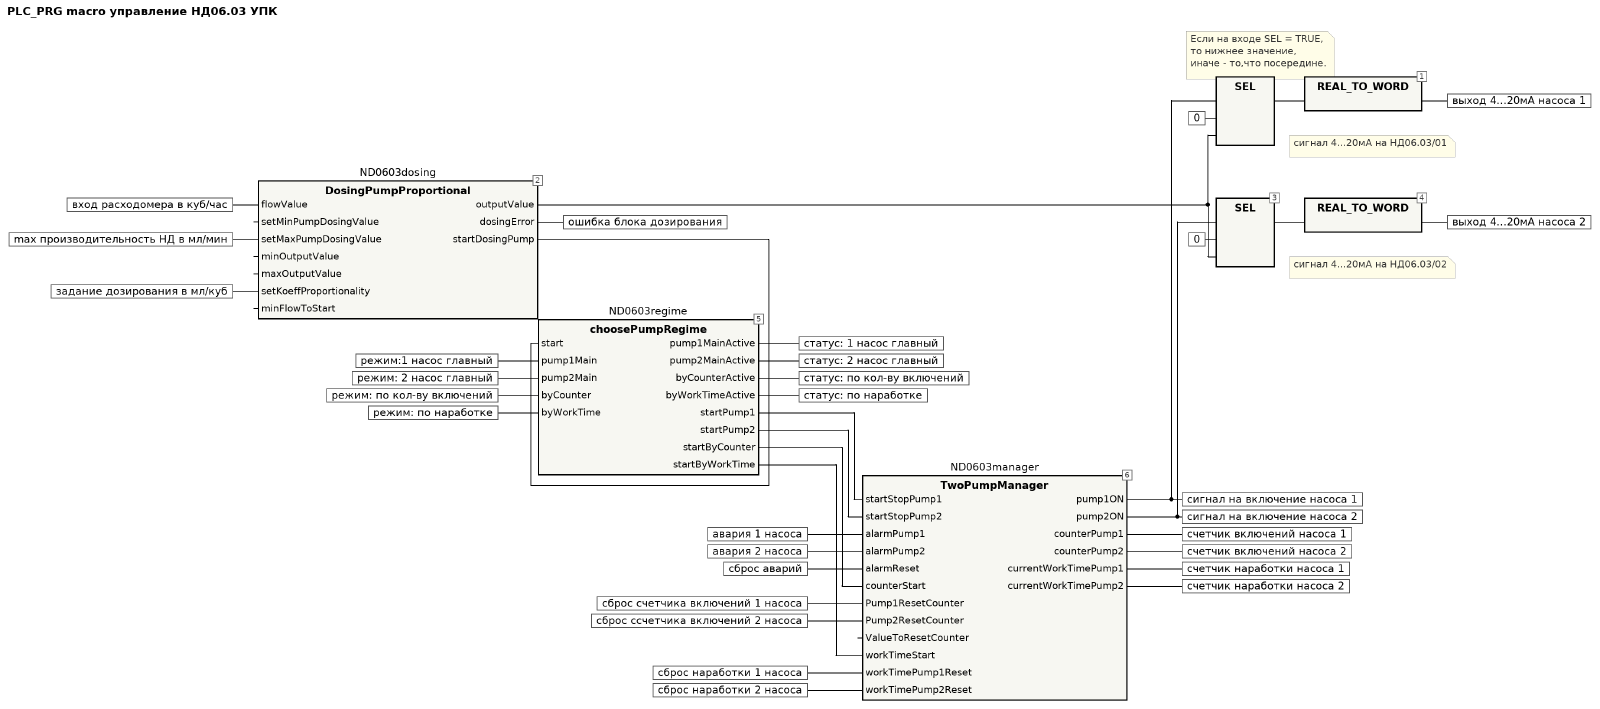
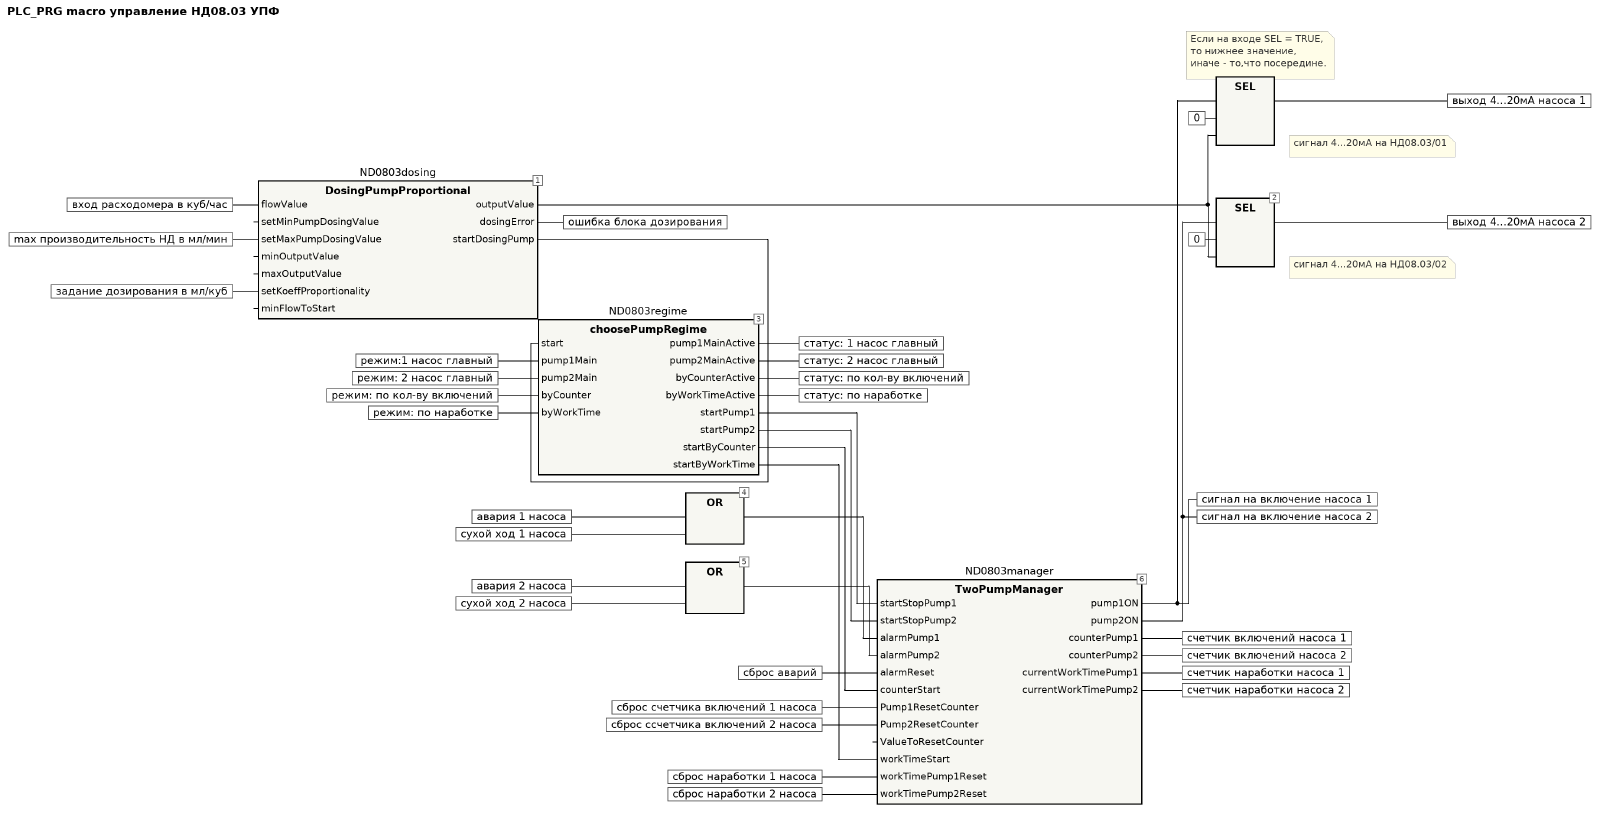
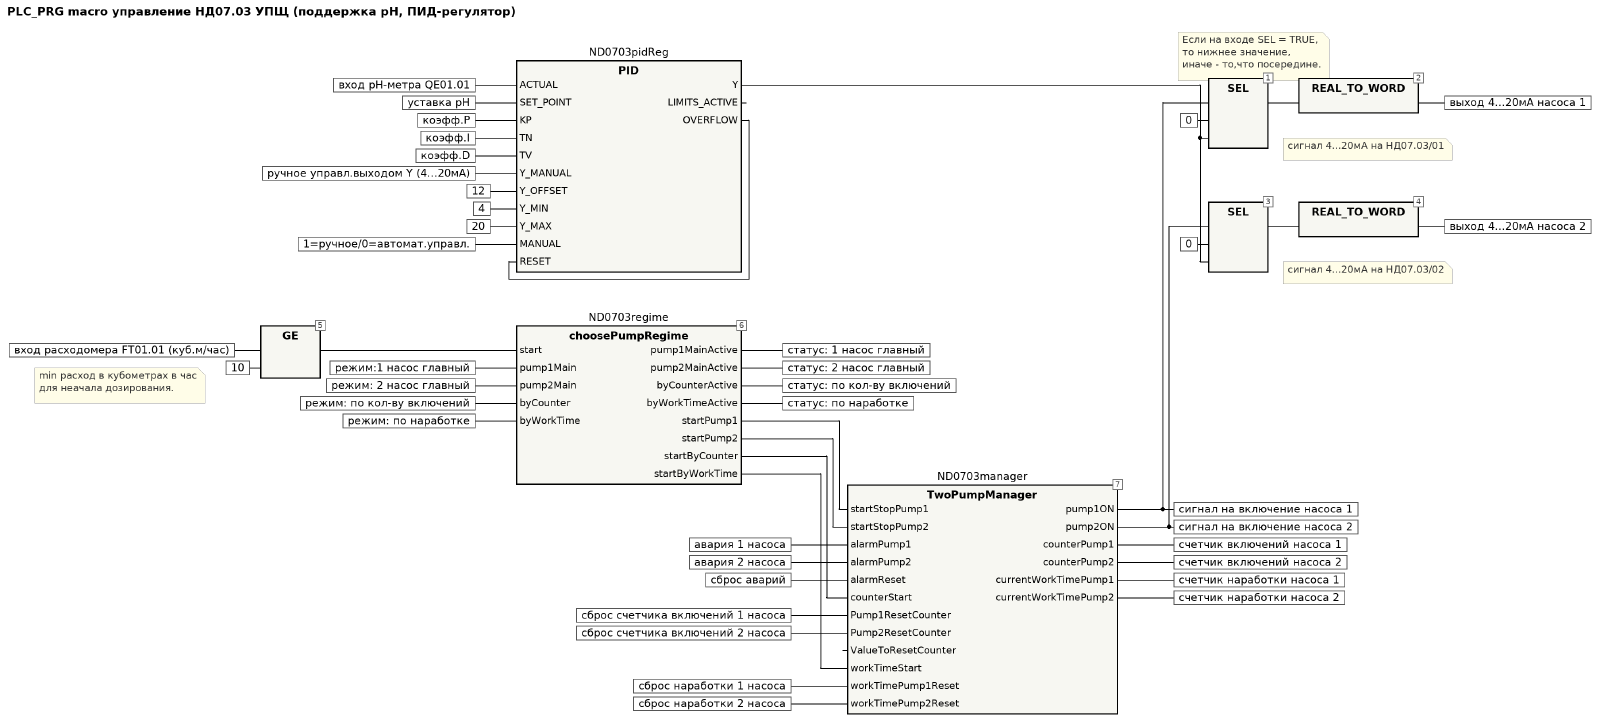
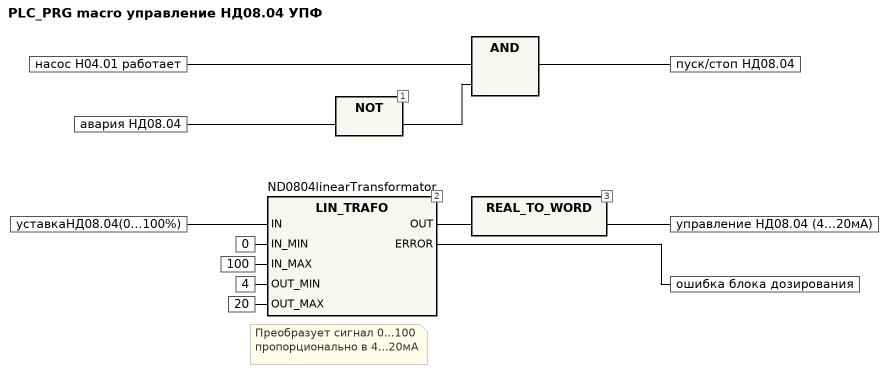
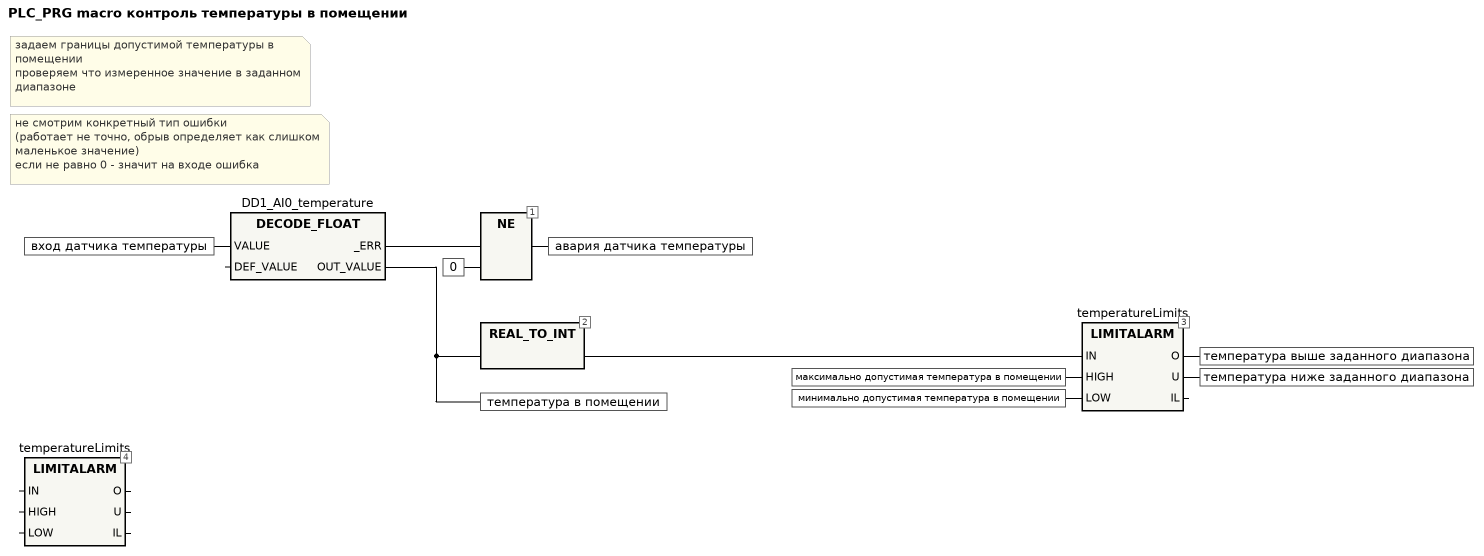
_CFC_ (* Continuous Function Chart, elements in execution order *)
(* рН-метр QE01.02 на входе, / диапазон 0...14 *)
(* авария входа рН-метра QE01.01 *)
(* авария входа расходомера FT01.02 *)
(* расходомер FT01.01 на входе, / диапазон 0...600куб/час *)
(* авария НД08.04 *)
(* управление 4...20мА НД08.03/01 *)
(* пуск/стоп НД08.03/01 *)
(* пуск/стоп НД08.03/02 *)
(* управление 4...20мА НД08.03/02 *)
(* авария привода НД08.03/01 *)
(* авария привода НД08.03/02 *)
(* авария НД07.03/01 *)
(* авария НД07.03/02 *)
(* управление 4...20мА НД07.03/01 *)
(* управление 4...20мА НД07.03/02 *)
(* пуск/стоп НД07.03/01 *)
(* пуск/стоп НД07.03/02 *)
(* авария НД07.03/01 *)
(* авария НД07.03/02 *)
(* авария НД06.03/01 *)
(* авария НД06.03/02 *)
(* авария НД06.02/01 *)
(* авария НД06.02/02 *)
(* авария НД05.02/01 *)
(* авария НД05.02/02 *)
(* управление 4...20мА НД06.03/01 *)
(* пуск/стоп НД06.03/01 *)
(* пуск/стоп НД06.03/02 *)
(* управление 4...20мА НД06.03/02 *)
(* авария НД06.03/01 *)
(* авария НД06.03/02 *)
(* управление 4...20мА НД06.02/01 *)
(* пуск/стоп НД06.02/01 *)
(* пуск/стоп НД06.02/02 *)
(* управление 4...20мА НД06.02/02 *)
(* авария НД06.02/01 *)
(* авария НД06.02/02 *)
(* ошибка блока дозирования НД05.02 *)
(* авария входа датчика температуры *)
(* лампа АВАРИЯ *)
(* датчик температуры в помещении / диапазон: 0...+100С *)
(* управление 4...20мА НД05.02/01 *)
(* пуск/стоп НД05.02/01 *)
(* авария НД05.02/01 *)
(* авария НД05.02/02 *)
(* пуск/стоп НД05.02/02 *)
(* управление 4...20мА НД05.02/02 *)
(* АВАРИИ *)
(* авария привода НД08.03/01 *)
(* авария привода НД08.03/02 *)
(* авария НД08.04 *)
(* насос Н04.01 работает *)
(* пуск/стоп НД08.04 *)
(* управление 4...20мА НД08.04 *)
(* авария входа расходомера FT01.01 *)
(* расходомер FT01.02 на входе, / диапазон 0...600куб/час *)
(* рН-метр QE01.01 на входе, / диапазон 0...14 *)
(* авария входа рН-метра QE01.02 *)
(* сухой ход НД08.03/01 *)
(* сухой ход НД08.03/02 *)
(* сухой ход НД08.03/01 *)
(* сухой ход НД08.03/02 *)
(* LSA01.02 перелив ОГМ01.04 *)
(* Инициализирует требуемые булевые переменные / в момент старта выполнения программы. *)
#0 rTrigStartInitializer:R_TRIG(CLK: TRUE)
#1 startInitializer <= #0.Q
#2 MACRO контроль аналогового входа DD1_AI1(pin 1 "вход": DD1_AI1)
	(* Не смотрим конкретную ошибку, / определяем,что вход неисправен без расшифровки. *)
	#3 DD1_AI1_FT0101:DECODE_FLOAT(VALUE: pin 1, DEF_VALUE: -)
	#4 NE(#3._ERR, 0)
	out 2 "авария" <= #4
	out 1 "выход" <= #3.OUT_VALUE
END_MACRO
#5 DD1_AI1_FT0101value <= #2.out 1
#6 DD1_AI1_error <= #2.out 2
#7 MACRO контроль аналогового входа DD1_AI2(pin 1 "вход": DD1_AI2)
	(* Не смотрим конкретную ошибку, / определяем,что вход неисправен без расшифровки. *)
	#8 DD1_AI2_FT0102:DECODE_FLOAT(VALUE: pin 1, DEF_VALUE: -)
	#9 NE(#8._ERR, 0)
	out 2 "авария" <= #9
	out 1 "выход" <= #8.OUT_VALUE
END_MACRO
#10 DD1_AI2_FT0102value <= #7.out 1
#11 DD1_AI2_error <= #7.out 2
#12 MACRO контроль аналогового входа DD1_AI3(pin 1 "вход": DD1_AI3)
	(* Не смотрим конкретную ошибку, / определяем,что вход неисправен без расшифровки. *)
	#13 DD1_AI3_QE0101:DECODE_FLOAT(VALUE: pin 1, DEF_VALUE: -)
	#14 NE(#13._ERR, 0)
	out 2 "авария" <= #14
	out 1 "выход" <= #13.OUT_VALUE
END_MACRO
#15 DD1_AI3_QE0101value <= #12.out 1
#16 DD1_AI3_error <= #12.out 2
#17 OR(DD1_AI0_error, alarmHighTemperature, alarmLowTemperature, ND0502dosingError, DD6_DI.0, DD6_DI.1, ND0502dosingError, DD6_DI.2, DD6_DI.3, ND0602dosingError, DD6_DI.4, DD6_DI.5, ND0603dosingError, DD6_DI.6, DD6_DI.7, ND0803dosingError, DD5_DI.12, DD5_DI.13, DD1_DI6, DD1_DI7, DD6_DI.16, ND0804dosingError, DD1_AI1_error, DD1_AI2_error, DD1_AI3_error, DD1_AI4_error, DD6_DI.11, N010501alarm, N010502alarm)
#18 DD1_DO11 <= #17
#19 MACRO управление НД06.02 УПК(pin 1 "вход расходомера в куб/час": DD1_AI2_FT0102value, pin 2 "max производительность НД в мл/мин": ND0602setMaxDosVal, pin 3 "задание дозирования в мл/куб": ND0602setKoefProp, pin 4 "режим:1 насос главный": ND0602regimeP1M, pin 5 "режим: 2 насос главный": ND0602regimeP2M, pin 6 "режим: по наработке": ND0602regimeByWT, pin 7 "режим: по кол-ву включений": ND0602regimeByC, pin 8 "авария 1 насоса": DD6_DI.2, pin 9 "авария 2 насоса": DD6_DI.3, pin 10 "сброс аварий": alarmReset, pin 11 "сброс счетчика включений 1 насоса": ND0602resetCountP1, pin 12 "сброс ссчетчика включений 2 насоса": ND0602resetCountP2, pin 13 "сброс наработки 1 насоса": ND0602resetWorkTimeP1, pin 14 "сброс наработки 2 насоса": ND0602resetWorkTimeP2)
	(* сигнал 4...20мА на НД06.02/02 *)
	(* сигнал 4...20мА на НД06.02/01 *)
	(* Если на входе SEL = TRUE, / то нижнее значение, / иначе - то,что посередине. *)
	#20 SEL(#26.pump1ON, 0, #22.outputValue)
	#21 REAL_TO_WORD(#20)
	out 6 "выход 4...20мА насоса 1" <= #21
	#22 ND0602dosing:DosingPumpProportional(flowValue: pin 1, setMinPumpDosingValue: -, setMaxPumpDosingValue: pin 2, minOutputValue: -, maxOutputValue: -, setKoeffProportionality: pin 3, minFlowToStart: -)
	out 1 "ошибка блока дозирования" <= #22.dosingError
	#23 SEL(#26.pump2ON, 0, #22.outputValue)
	#24 REAL_TO_WORD(#23)
	out 7 "выход 4...20мА насоса 2" <= #24
	#25 ND0602regime:choosePumpRegime(start: #22.startDosingPump, pump1Main: pin 4, pump2Main: pin 5, byCounter: pin 7, byWorkTime: pin 6)
	out 2 "статус: 1 насос главный" <= #25.pump1MainActive
	out 3 "статус: 2 насос главный" <= #25.pump2MainActive
	out 4 "статус: по кол-ву включений" <= #25.byCounterActive
	out 5 "статус: по наработке" <= #25.byWorkTimeActive
	#26 ND0602manager:TwoPumpManager(startStopPump1: #25.startPump1, startStopPump2: #25.startPump2, alarmPump1: pin 8, alarmPump2: pin 9, alarmReset: pin 10, counterStart: #25.startByCounter, Pump1ResetCounter: pin 11, Pump2ResetCounter: pin 12, ValueToResetCounter: -, workTimeStart: #25.startByWorkTime, workTimePump1Reset: pin 13, workTimePump2Reset: pin 14)
	out 12 "сигнал на включение насоса 1" <= #26.pump1ON
	out 13 "сигнал на включение насоса 2" <= #26.pump2ON
	out 8 "счетчик включений насоса 1" <= #26.counterPump1
	out 9 "счетчик включений насоса 2" <= #26.counterPump2
	out 10 "счетчик наработки насоса 1" <= #26.currentWorkTimePump1
	out 11 "счетчик наработки насоса 2" <= #26.currentWorkTimePump2
END_MACRO
#27 ND0602dosingError <= #19.out 1
#28 ND0602statRegimeP1M <= #19.out 2
#29 ND0602statRegimeP2M <= #19.out 3
#30 ND0602statRegimeByC <= #19.out 4
#31 ND0602statRegimeByWT <= #19.out 5
#32 DD10_AO1 <= #19.out 6
#33 DD10_AO2 <= #19.out 7
#34 ND0602counterP1 <= #19.out 8
#35 ND0602counterP2 <= #19.out 9
#36 ND0602workTimeP1 <= #19.out 10
#37 ND0602workTimeP2 <= #19.out 11
#38 DD4_DO.6 <= #19.out 12
#39 DD4_DO.7 <= #19.out 13
#40 MACRO контроль аналогового входа DD1_AI4(pin 1 "вход": DD1_AI4)
	(* Не смотрим конкретную ошибку, / определяем,что вход неисправен без расшифровки. *)
	#41 DD1_AI4_QE0102:DECODE_FLOAT(VALUE: pin 1, DEF_VALUE: -)
	#42 NE(#41._ERR, 0)
	out 2 "авария" <= #42
	out 1 "выход" <= #41.OUT_VALUE
END_MACRO
#43 DD1_AI4_QE0102value <= #40.out 1
#44 DD1_AI4_error <= #40.out 2
#45 MACRO управление НД05.02 УПГ(pin 1 "вход расходомера в куб/час": DD1_AI1_FT0101value, pin 2 "max производительность НД в мл/мин": ND0502setMaxDosVal, pin 3 "задание дозирования в мл/куб": ND0502setKoefProp, pin 4 "режим:1 насос главный": ND0502regimeP1M, pin 5 "режим: 2 насос главный": ND0502regimeP2M, pin 6 "режим: по наработке": ND0502regimeByWT, pin 7 "режим: по кол-ву включений": ND0502regimeByC, pin 8 "авария 1 насоса": DD6_DI.0, pin 9 "авария 2 насоса": DD6_DI.1, pin 10 "сброс аварий": alarmReset, pin 11 "сброс счетчика включений 1 насоса": ND0502resetCountP1, pin 12 "сброс ссчетчика включений 2 насоса": ND0502resetCountP2, pin 13 "сброс наработки 1 насоса": ND0502resetWorkTimeP1, pin 14 "сброс наработки 2 насоса": ND0502resetWorkTimeP2)
	(* сигнал 4...20мА на НД05.02/02 *)
	(* сигнал 4...20мА на НД05.02/01 *)
	(* Если на входе SEL = TRUE, / то нижнее значение, / иначе - то,что посередине. *)
	#46 SEL(#51.pump1ON, 0, #47.outputValue)
	out 6 "выход 4...20мА насоса 1" <= #46
	#47 ND0502dosing:DosingPumpProportional(flowValue: pin 1, setMinPumpDosingValue: -, setMaxPumpDosingValue: pin 2, minOutputValue: -, maxOutputValue: -, setKoeffProportionality: pin 3, minFlowToStart: -)
	out 1 "ошибка блока дозирования" <= #47.dosingError
	#48 SEL(#51.pump2ON, 0, #47.outputValue)
	#49 REAL_TO_WORD(#48)
	out 7 "выход 4...20мА насоса 2" <= #49
	#50 ND0502regime:choosePumpRegime(start: #47.startDosingPump, pump1Main: pin 4, pump2Main: pin 5, byCounter: pin 7, byWorkTime: pin 6)
	out 2 "статус: 1 насос главный" <= #50.pump1MainActive
	out 3 "статус: 2 насос главный" <= #50.pump2MainActive
	out 4 "статус: по кол-ву включений" <= #50.byCounterActive
	out 5 "статус: по наработке" <= #50.byWorkTimeActive
	#51 ND0502manager:TwoPumpManager(startStopPump1: #50.startPump1, startStopPump2: #50.startPump2, alarmPump1: pin 8, alarmPump2: pin 9, alarmReset: pin 10, counterStart: #50.startByCounter, Pump1ResetCounter: pin 11, Pump2ResetCounter: pin 12, ValueToResetCounter: -, workTimeStart: #50.startByWorkTime, workTimePump1Reset: pin 13, workTimePump2Reset: pin 14)
	out 12 "сигнал на включение насоса 1" <= #51.pump1ON
	out 13 "сигнал на включение насоса 2" <= #51.pump2ON
	out 8 "счетчик включений насоса 1" <= #51.counterPump1
	out 9 "счетчик включений насоса 2" <= #51.counterPump2
	out 10 "счетчик наработки насоса 1" <= #51.currentWorkTimePump1
	out 11 "счетчик наработки насоса 2" <= #51.currentWorkTimePump2
END_MACRO
#52 ND0502dosingError <= #45.out 1
#53 ND0502statRegimeP1M <= #45.out 2
#54 ND0502statRegimeP2M <= #45.out 3
#55 ND0502statRegimeByC <= #45.out 4
#56 ND0502statRegimeByWT <= #45.out 5
#57 DD1_AO3 <= #45.out 6
#58 DD10_AO0 <= #45.out 7
#59 ND0502counterP1 <= #45.out 8
#60 ND0502counterP2 <= #45.out 9
#61 ND0502workTimeP1 <= #45.out 10
#62 ND0502workTimeP2 <= #45.out 11
#63 DD4_DO.4 <= #45.out 12
#64 DD4_DO.5 <= #45.out 13
#65 MACRO управление НД06.03 УПК(pin 1 "вход расходомера в куб/час": DD1_AI1_FT0101value, pin 2 "max производительность НД в мл/мин": ND0603setMaxDosVal, pin 3 "задание дозирования в мл/куб": ND0603setKoefProp, pin 4 "режим:1 насос главный": ND0603regimeP1M, pin 5 "режим: 2 насос главный": ND0603regimeP2M, pin 6 "режим: по наработке": ND0603regimeByWT, pin 7 "режим: по кол-ву включений": ND0603regimeByC, pin 8 "авария 1 насоса": DD6_DI.4, pin 9 "авария 2 насоса": DD6_DI.5, pin 10 "сброс аварий": alarmReset, pin 11 "сброс счетчика включений 1 насоса": ND0603resetCountP1, pin 12 "сброс ссчетчика включений 2 насоса": ND0603resetCountP2, pin 13 "сброс наработки 1 насоса": ND0603resetWorkTimeP1, pin 14 "сброс наработки 2 насоса": ND0603resetWorkTimeP2)
	(* сигнал 4...20мА на НД06.03/02 *)
	(* сигнал 4...20мА на НД06.03/01 *)
	(* Если на входе SEL = TRUE, / то нижнее значение, / иначе - то,что посередине. *)
	#66 SEL(#72.pump1ON, 0, #68.outputValue)
	#67 REAL_TO_WORD(#66)
	out 6 "выход 4...20мА насоса 1" <= #67
	#68 ND0603dosing:DosingPumpProportional(flowValue: pin 1, setMinPumpDosingValue: -, setMaxPumpDosingValue: pin 2, minOutputValue: -, maxOutputValue: -, setKoeffProportionality: pin 3, minFlowToStart: -)
	out 1 "ошибка блока дозирования" <= #68.dosingError
	#69 SEL(#72.pump2ON, 0, #68.outputValue)
	#70 REAL_TO_WORD(#69)
	out 7 "выход 4...20мА насоса 2" <= #70
	#71 ND0603regime:choosePumpRegime(start: #68.startDosingPump, pump1Main: pin 4, pump2Main: pin 5, byCounter: pin 7, byWorkTime: pin 6)
	out 2 "статус: 1 насос главный" <= #71.pump1MainActive
	out 3 "статус: 2 насос главный" <= #71.pump2MainActive
	out 4 "статус: по кол-ву включений" <= #71.byCounterActive
	out 5 "статус: по наработке" <= #71.byWorkTimeActive
	#72 ND0603manager:TwoPumpManager(startStopPump1: #71.startPump1, startStopPump2: #71.startPump2, alarmPump1: pin 8, alarmPump2: pin 9, alarmReset: pin 10, counterStart: #71.startByCounter, Pump1ResetCounter: pin 11, Pump2ResetCounter: pin 12, ValueToResetCounter: -, workTimeStart: #71.startByWorkTime, workTimePump1Reset: pin 13, workTimePump2Reset: pin 14)
	out 12 "сигнал на включение насоса 1" <= #72.pump1ON
	out 13 "сигнал на включение насоса 2" <= #72.pump2ON
	out 8 "счетчик включений насоса 1" <= #72.counterPump1
	out 9 "счетчик включений насоса 2" <= #72.counterPump2
	out 10 "счетчик наработки насоса 1" <= #72.currentWorkTimePump1
	out 11 "счетчик наработки насоса 2" <= #72.currentWorkTimePump2
END_MACRO
#73 ND0603dosingError <= #65.out 1
#74 ND0603statRegimeP1M <= #65.out 2
#75 ND0603statRegimeP2M <= #65.out 3
#76 ND0603statRegimeByC <= #65.out 4
#77 ND0603statRegimeByWT <= #65.out 5
#78 DD10_AO3 <= #65.out 6
#79 DD10_AO4 <= #65.out 7
#80 ND0603counterP1 <= #65.out 8
#81 ND0603counterP2 <= #65.out 9
#82 ND0603workTimeP1 <= #65.out 10
#83 ND0603workTimeP2 <= #65.out 11
#84 DD4_DO.8 <= #65.out 12
#85 DD4_DO.9 <= #65.out 13
#86 MACRO управление НД08.03 УПФ(pin 1 "вход расходомера в куб/час": DD1_AI1_FT0101value, pin 2 "max производительность НД в мл/мин": ND0803setMaxDosVal, pin 3 "задание дозирования в мл/куб": ND0803setKoefProp, pin 4 "режим:1 насос главный": ND0803regimeP1M, pin 5 "режим: 2 насос главный": ND0803regimeP2M, pin 6 "режим: по наработке": ND0803regimeByWT, pin 7 "режим: по кол-ву включений": ND0803regimeByC, pin 8 "авария 1 насоса": DD5_DI.12, pin 9 "авария 2 насоса": DD5_DI.13, pin 10 "сброс аварий": alarmReset, pin 11 "сброс счетчика включений 1 насоса": ND0803resetCountP1, pin 12 "сброс ссчетчика включений 2 насоса": ND0803resetCountP2, pin 13 "сброс наработки 1 насоса": ND0803resetWorkTimeP1, pin 14 "сброс наработки 2 насоса": ND0803resetWorkTimeP2, pin 15 "сухой ход 1 насоса": DD1_DI6, pin 16 "сухой ход 2 насоса": DD1_DI7)
	(* сигнал 4...20мА на НД08.03/02 *)
	(* сигнал 4...20мА на НД08.03/01 *)
	(* Если на входе SEL = TRUE, / то нижнее значение, / иначе - то,что посередине. *)
	#87 SEL(#93.pump1ON, 0, #88.outputValue)
	out 6 "выход 4...20мА насоса 1" <= #87
	#88 ND0803dosing:DosingPumpProportional(flowValue: pin 1, setMinPumpDosingValue: -, setMaxPumpDosingValue: pin 2, minOutputValue: -, maxOutputValue: -, setKoeffProportionality: pin 3, minFlowToStart: -)
	out 1 "ошибка блока дозирования" <= #88.dosingError
	#89 SEL(#93.pump2ON, 0, #88.outputValue)
	out 7 "выход 4...20мА насоса 2" <= #89
	#90 ND0803regime:choosePumpRegime(start: #88.startDosingPump, pump1Main: pin 4, pump2Main: pin 5, byCounter: pin 7, byWorkTime: pin 6)
	out 2 "статус: 1 насос главный" <= #90.pump1MainActive
	out 3 "статус: 2 насос главный" <= #90.pump2MainActive
	out 4 "статус: по кол-ву включений" <= #90.byCounterActive
	out 5 "статус: по наработке" <= #90.byWorkTimeActive
	out 12 "сигнал на включение насоса 1" <= #93.pump1ON
	#91 OR(pin 8, pin 15)
	out 13 "сигнал на включение насоса 2" <= #93.pump2ON
	#92 OR(pin 9, pin 16)
	#93 ND0803manager:TwoPumpManager(startStopPump1: #90.startPump1, startStopPump2: #90.startPump2, alarmPump1: #91, alarmPump2: #92, alarmReset: pin 10, counterStart: #90.startByCounter, Pump1ResetCounter: pin 11, Pump2ResetCounter: pin 12, ValueToResetCounter: -, workTimeStart: #90.startByWorkTime, workTimePump1Reset: pin 13, workTimePump2Reset: pin 14)
	out 8 "счетчик включений насоса 1" <= #93.counterPump1
	out 9 "счетчик включений насоса 2" <= #93.counterPump2
	out 10 "счетчик наработки насоса 1" <= #93.currentWorkTimePump1
	out 11 "счетчик наработки насоса 2" <= #93.currentWorkTimePump2
END_MACRO
#94 ND0803dosingError <= #86.out 1
#95 ND0803statRegimeP1M <= #86.out 2
#96 ND0803statRegimeP2M <= #86.out 3
#97 ND0803statRegimeByC <= #86.out 4
#98 ND0803statRegimeByWT <= #86.out 5
#99 DD1_AO1 <= #86.out 6
#100 DD1_AO2 <= #86.out 7
#101 ND0803counterP1 <= #86.out 8
#102 ND0803counterP2 <= #86.out 9
#103 ND0803workTimeP1 <= #86.out 10
#104 ND0803workTimeP2 <= #86.out 11
#105 DD1_DO3 <= #86.out 12
#106 DD1_DO4 <= #86.out 13
#107 MACRO управление НД07.03 УПЩ (поддержка рН, ПИД-регулятор)(pin 1 "вход рН-метра QE01.01": DD1_AI3_QE0101value, pin 2 "уставка рН": ND0703pHsetValue, pin 3 "режим:1 насос главный": ND0703regimeP1M, pin 4 "режим: 2 насос главный": ND0703regimeP2M, pin 5 "режим: по наработке": ND0703regimeByWT, pin 6 "режим: по кол-ву включений": ND0703regimeByC, pin 7 "авария 1 насоса": DD6_DI.6, pin 8 "авария 2 насоса": DD6_DI.7, pin 9 "сброс аварий": alarmReset, pin 10 "сброс счетчика включений 1 насоса": ND0703resetCountP1, pin 11 "сброс счетчика включений 2 насоса": ND0703resetCountP2, pin 12 "сброс наработки 1 насоса": ND0703resetWorkTimeP1, pin 13 "сброс наработки 2 насоса": ND0703resetWorkTimeP2, pin 14 "ручное управл.выходом Y (4...20мА)": ND0703YoutManual, pin 15 "1=ручное/0=автомат.управл.": ND0703YmanAuto, pin 16 "вход расходомера FT01.01 (куб.м/час)": DD1_AI1_FT0101value, pin 17 "коэфф.I": ND0703koeffI, pin 18 "коэфф.D": ND0703koeffD, pin 19 "коэфф.Р": ND0703koeffP)
	(* сигнал 4...20мА на НД07.03/02 *)
	(* сигнал 4...20мА на НД07.03/01 *)
	(* Если на входе SEL = TRUE, / то нижнее значение, / иначе - то,что посередине. *)
	(* min расход в кубометрах в час / для неачала дозирования. *)
	#108 ND0703pidReg:PID(ACTUAL: pin 1, SET_POINT: pin 2, KP: pin 19, TN: pin 17, TV: pin 18, Y_MANUAL: pin 14, Y_OFFSET: 12, Y_MIN: 4, Y_MAX: 20, MANUAL: pin 15, RESET: #108.OVERFLOW)
	#109 SEL(#115.pump1ON, 0, #108.Y)
	#110 REAL_TO_WORD(#109)
	out 5 "выход 4...20мА насоса 1" <= #110
	#111 SEL(#115.pump2ON, 0, #108.Y)
	#112 REAL_TO_WORD(#111)
	out 6 "выход 4...20мА насоса 2" <= #112
	#113 GE(pin 16, 10)
	#114 ND0703regime:choosePumpRegime(start: #113, pump1Main: pin 3, pump2Main: pin 4, byCounter: pin 6, byWorkTime: pin 5)
	out 1 "статус: 1 насос главный" <= #114.pump1MainActive
	out 2 "статус: 2 насос главный" <= #114.pump2MainActive
	out 3 "статус: по кол-ву включений" <= #114.byCounterActive
	out 4 "статус: по наработке" <= #114.byWorkTimeActive
	#115 ND0703manager:TwoPumpManager(startStopPump1: #114.startPump1, startStopPump2: #114.startPump2, alarmPump1: pin 7, alarmPump2: pin 8, alarmReset: pin 9, counterStart: #114.startByCounter, Pump1ResetCounter: pin 10, Pump2ResetCounter: pin 11, ValueToResetCounter: -, workTimeStart: #114.startByWorkTime, workTimePump1Reset: pin 12, workTimePump2Reset: pin 13)
	out 11 "сигнал на включение насоса 1" <= #115.pump1ON
	out 12 "сигнал на включение насоса 2" <= #115.pump2ON
	out 7 "счетчик включений насоса 1" <= #115.counterPump1
	out 8 "счетчик включений насоса 2" <= #115.counterPump2
	out 9 "счетчик наработки насоса 1" <= #115.currentWorkTimePump1
	out 10 "счетчик наработки насоса 2" <= #115.currentWorkTimePump2
END_MACRO
#116 ND0703statRegimeP1M <= #107.out 1
#117 ND0703statRegimeP2M <= #107.out 2
#118 ND0703statRegimeByC <= #107.out 3
#119 ND0703statRegimeByWT <= #107.out 4
#120 DD10_AO5 <= #107.out 5
#121 DD10_AO6 <= #107.out 6
#122 ND0703counterP1 <= #107.out 7
#123 ND0703counterP2 <= #107.out 8
#124 ND0703workTimeP1 <= #107.out 9
#125 ND0703workTimeP2 <= #107.out 10
#126 DD4_DO.10 <= #107.out 11
#127 DD4_DO.11 <= #107.out 12
#128 MACRO управление НД08.04 УПФ(pin 1 "насос Н04.01 работает": DD7_DI.13, pin 2 "авария НД08.04": DD6_DI.16, pin 3 "уставкаНД08.04(0...100%)": ND0804doseValue)
	(* Преобразует сигнал 0...100 / пропорционально в 4...20мА *)
	#129 AND(pin 1, #130)
	out 1 "пуск/стоп НД08.04" <= #129
	#130 NOT(pin 2)
	#131 ND0804linearTransformator:LIN_TRAFO(IN: pin 3, IN_MIN: 0, IN_MAX: 100, OUT_MIN: 4, OUT_MAX: 20)
	#132 REAL_TO_WORD(#131.OUT)
	out 2 "управление НД08.04 (4...20мА)" <= #132
	out 3 "ошибка блока дозирования" <= #131.ERROR
END_MACRO
#133 DD4_DO.12 <= #128.out 1
#134 DD10_AO7 <= #128.out 2
#135 ND0804dosingError <= #128.out 3
#136 MACRO контроль температуры в помещении(pin 1 "вход датчика температуры": DD1_AI0, pin 2 "минимально допустимая температура в помещении": maxTemperature, pin 3 "максимально допустимая температура в помещении": minTemperature)
	(* задаем границы допустимой температуры в помещении / проверяем что измеренное значение в заданном диапазоне *)
	(* не смотрим конкретный тип ошибки / (работает не точно, обрыв определяет как слишком маленькое значение) / если не равно 0 - значит на входе ошибка *)
	#137 DD1_AI0_temperature:DECODE_FLOAT(VALUE: pin 1, DEF_VALUE: -)
	#138 NE(#137._ERR, 0)
	out 2 "авария датчика температуры" <= #138
	out 1 "температура в помещении" <= #137.OUT_VALUE
	#139 REAL_TO_INT(#137.OUT_VALUE)
	#140 temperatureLimits:LIMITALARM(IN: #139, HIGH: pin 3, LOW: pin 2)
	out 3 "температура выше заданного диапазона" <= #140.O
	out 4 "температура ниже заданного диапазона" <= #140.U
	#141 temperatureLimits:LIMITALARM(IN: -, HIGH: -, LOW: -)
END_MACRO
#142 temperatureValue <= #136.out 1
#143 DD1_AI0_error <= #136.out 2
#144 alarmHighTemperature <= #136.out 3
#145 alarmLowTemperature <= #136.out 4
#146 tempTwoPumpOneDriveManager:TwoPumpOneDriveManager(startStopPump1: temp1, startStopPump2: temp2, alarmPump1: temp3, alarmPump2: temp4, alarmReset: temp5, counterStart: temp6, Pump1ResetCounter: temp7, Pump2ResetCounter: temp8, ValueToResetCounter: -, workTimeStart: temp9, workTimePump1Reset: temp10, workTimePump2Reset: temp11, timeKM1off: -, timeKM23DelayON: -, timeKM23offDelay: -, timeReadyToStartDelay: -)
#147 temp12 <= #146.counterPump1
#148 temp13 <= #146.counterPump2
#149 temp14 <= #146.currentWorkTimePump1
#150 temp15 <= #146.currentWorkTimePump2
#151 temp16 <= #146.DriveKM
#152 temp17 <= #146.pump1KM
#153 temp18 <= #146.pump2KM
#154 temp19 <= #146.driveStart
_END_CFC_
(* the same logic as Structured Text *)
(* рН-метр QE01.02 на входе, / диапазон 0...14 *)
(* авария входа рН-метра QE01.01 *)
(* авария входа расходомера FT01.02 *)
(* расходомер FT01.01 на входе, / диапазон 0...600куб/час *)
(* авария НД08.04 *)
(* управление 4...20мА НД08.03/01 *)
(* пуск/стоп НД08.03/01 *)
(* пуск/стоп НД08.03/02 *)
(* управление 4...20мА НД08.03/02 *)
(* авария привода НД08.03/01 *)
(* авария привода НД08.03/02 *)
(* авария НД07.03/01 *)
(* авария НД07.03/02 *)
(* управление 4...20мА НД07.03/01 *)
(* управление 4...20мА НД07.03/02 *)
(* пуск/стоп НД07.03/01 *)
(* пуск/стоп НД07.03/02 *)
(* авария НД07.03/01 *)
(* авария НД07.03/02 *)
(* авария НД06.03/01 *)
(* авария НД06.03/02 *)
(* авария НД06.02/01 *)
(* авария НД06.02/02 *)
(* авария НД05.02/01 *)
(* авария НД05.02/02 *)
(* управление 4...20мА НД06.03/01 *)
(* пуск/стоп НД06.03/01 *)
(* пуск/стоп НД06.03/02 *)
(* управление 4...20мА НД06.03/02 *)
(* авария НД06.03/01 *)
(* авария НД06.03/02 *)
(* управление 4...20мА НД06.02/01 *)
(* пуск/стоп НД06.02/01 *)
(* пуск/стоп НД06.02/02 *)
(* управление 4...20мА НД06.02/02 *)
(* авария НД06.02/01 *)
(* авария НД06.02/02 *)
(* ошибка блока дозирования НД05.02 *)
(* авария входа датчика температуры *)
(* лампа АВАРИЯ *)
(* датчик температуры в помещении / диапазон: 0...+100С *)
(* управление 4...20мА НД05.02/01 *)
(* пуск/стоп НД05.02/01 *)
(* авария НД05.02/01 *)
(* авария НД05.02/02 *)
(* пуск/стоп НД05.02/02 *)
(* управление 4...20мА НД05.02/02 *)
(* АВАРИИ *)
(* авария привода НД08.03/01 *)
(* авария привода НД08.03/02 *)
(* авария НД08.04 *)
(* насос Н04.01 работает *)
(* пуск/стоп НД08.04 *)
(* управление 4...20мА НД08.04 *)
(* авария входа расходомера FT01.01 *)
(* расходомер FT01.02 на входе, / диапазон 0...600куб/час *)
(* рН-метр QE01.01 на входе, / диапазон 0...14 *)
(* авария входа рН-метра QE01.02 *)
(* сухой ход НД08.03/01 *)
(* сухой ход НД08.03/02 *)
(* сухой ход НД08.03/01 *)
(* сухой ход НД08.03/02 *)
(* LSA01.02 перелив ОГМ01.04 *)
(* Инициализирует требуемые булевые переменные / в момент старта выполнения программы. *)
rTrigStartInitializer(CLK := TRUE);
startInitializer := rTrigStartInitializer.Q;
(* macro контроль аналогового входа DD1_AI1 *)
(* Не смотрим конкретную ошибку, / определяем,что вход неисправен без расшифровки. *)
DD1_AI1_FT0101(VALUE := DD1_AI1);
DD1_AI1_FT0101value := DD1_AI1_FT0101.OUT_VALUE;
DD1_AI1_error := DD1_AI1_FT0101._ERR <> 0;
(* macro контроль аналогового входа DD1_AI2 *)
(* Не смотрим конкретную ошибку, / определяем,что вход неисправен без расшифровки. *)
DD1_AI2_FT0102(VALUE := DD1_AI2);
DD1_AI2_FT0102value := DD1_AI2_FT0102.OUT_VALUE;
DD1_AI2_error := DD1_AI2_FT0102._ERR <> 0;
(* macro контроль аналогового входа DD1_AI3 *)
(* Не смотрим конкретную ошибку, / определяем,что вход неисправен без расшифровки. *)
DD1_AI3_QE0101(VALUE := DD1_AI3);
DD1_AI3_QE0101value := DD1_AI3_QE0101.OUT_VALUE;
DD1_AI3_error := DD1_AI3_QE0101._ERR <> 0;
DD1_DO11 := DD1_AI0_error OR alarmHighTemperature OR alarmLowTemperature OR ND0502dosingError OR DD6_DI.0 OR DD6_DI.1 OR ND0502dosingError OR DD6_DI.2 OR DD6_DI.3 OR ND0602dosingError OR DD6_DI.4 OR DD6_DI.5 OR ND0603dosingError OR DD6_DI.6 OR DD6_DI.7 OR ND0803dosingError OR DD5_DI.12 OR DD5_DI.13 OR DD1_DI6 OR DD1_DI7 OR DD6_DI.16 OR ND0804dosingError OR DD1_AI1_error OR DD1_AI2_error OR DD1_AI3_error OR DD1_AI4_error OR DD6_DI.11 OR N010501alarm OR N010502alarm;
(* macro управление НД06.02 УПК *)
(* сигнал 4...20мА на НД06.02/02 *)
(* сигнал 4...20мА на НД06.02/01 *)
(* Если на входе SEL = TRUE, / то нижнее значение, / иначе - то,что посередине. *)
_t977 := REAL_TO_WORD(SEL(ND0602manager.pump1ON, 0, ND0602dosing.outputValue));
ND0602dosing(flowValue := DD1_AI2_FT0102value, setMaxPumpDosingValue := ND0602setMaxDosVal, setKoeffProportionality := ND0602setKoefProp);
_t899 := REAL_TO_WORD(SEL(ND0602manager.pump2ON, 0, ND0602dosing.outputValue));
ND0602regime(start := ND0602dosing.startDosingPump, pump1Main := ND0602regimeP1M, pump2Main := ND0602regimeP2M, byCounter := ND0602regimeByC, byWorkTime := ND0602regimeByWT);
ND0602manager(startStopPump1 := ND0602regime.startPump1, startStopPump2 := ND0602regime.startPump2, alarmPump1 := DD6_DI.2, alarmPump2 := DD6_DI.3, alarmReset := alarmReset, counterStart := ND0602regime.startByCounter, Pump1ResetCounter := ND0602resetCountP1, Pump2ResetCounter := ND0602resetCountP2, workTimeStart := ND0602regime.startByWorkTime, workTimePump1Reset := ND0602resetWorkTimeP1, workTimePump2Reset := ND0602resetWorkTimeP2);
ND0602dosingError := ND0602dosing.dosingError;
ND0602statRegimeP1M := ND0602regime.pump1MainActive;
ND0602statRegimeP2M := ND0602regime.pump2MainActive;
ND0602statRegimeByC := ND0602regime.byCounterActive;
ND0602statRegimeByWT := ND0602regime.byWorkTimeActive;
DD10_AO1 := _t977;
DD10_AO2 := _t899;
ND0602counterP1 := ND0602manager.counterPump1;
ND0602counterP2 := ND0602manager.counterPump2;
ND0602workTimeP1 := ND0602manager.currentWorkTimePump1;
ND0602workTimeP2 := ND0602manager.currentWorkTimePump2;
DD4_DO.6 := ND0602manager.pump1ON;
DD4_DO.7 := ND0602manager.pump2ON;
(* macro контроль аналогового входа DD1_AI4 *)
(* Не смотрим конкретную ошибку, / определяем,что вход неисправен без расшифровки. *)
DD1_AI4_QE0102(VALUE := DD1_AI4);
DD1_AI4_QE0102value := DD1_AI4_QE0102.OUT_VALUE;
DD1_AI4_error := DD1_AI4_QE0102._ERR <> 0;
(* macro управление НД05.02 УПГ *)
(* сигнал 4...20мА на НД05.02/02 *)
(* сигнал 4...20мА на НД05.02/01 *)
(* Если на входе SEL = TRUE, / то нижнее значение, / иначе - то,что посередине. *)
_t831 := SEL(ND0502manager.pump1ON, 0, ND0502dosing.outputValue);
ND0502dosing(flowValue := DD1_AI1_FT0101value, setMaxPumpDosingValue := ND0502setMaxDosVal, setKoeffProportionality := ND0502setKoefProp);
_t801 := REAL_TO_WORD(SEL(ND0502manager.pump2ON, 0, ND0502dosing.outputValue));
ND0502regime(start := ND0502dosing.startDosingPump, pump1Main := ND0502regimeP1M, pump2Main := ND0502regimeP2M, byCounter := ND0502regimeByC, byWorkTime := ND0502regimeByWT);
ND0502manager(startStopPump1 := ND0502regime.startPump1, startStopPump2 := ND0502regime.startPump2, alarmPump1 := DD6_DI.0, alarmPump2 := DD6_DI.1, alarmReset := alarmReset, counterStart := ND0502regime.startByCounter, Pump1ResetCounter := ND0502resetCountP1, Pump2ResetCounter := ND0502resetCountP2, workTimeStart := ND0502regime.startByWorkTime, workTimePump1Reset := ND0502resetWorkTimeP1, workTimePump2Reset := ND0502resetWorkTimeP2);
ND0502dosingError := ND0502dosing.dosingError;
ND0502statRegimeP1M := ND0502regime.pump1MainActive;
ND0502statRegimeP2M := ND0502regime.pump2MainActive;
ND0502statRegimeByC := ND0502regime.byCounterActive;
ND0502statRegimeByWT := ND0502regime.byWorkTimeActive;
DD1_AO3 := _t831;
DD10_AO0 := _t801;
ND0502counterP1 := ND0502manager.counterPump1;
ND0502counterP2 := ND0502manager.counterPump2;
ND0502workTimeP1 := ND0502manager.currentWorkTimePump1;
ND0502workTimeP2 := ND0502manager.currentWorkTimePump2;
DD4_DO.4 := ND0502manager.pump1ON;
DD4_DO.5 := ND0502manager.pump2ON;
(* macro управление НД06.03 УПК *)
(* сигнал 4...20мА на НД06.03/02 *)
(* сигнал 4...20мА на НД06.03/01 *)
(* Если на входе SEL = TRUE, / то нижнее значение, / иначе - то,что посередине. *)
_t1027 := REAL_TO_WORD(SEL(ND0603manager.pump1ON, 0, ND0603dosing.outputValue));
ND0603dosing(flowValue := DD1_AI1_FT0101value, setMaxPumpDosingValue := ND0603setMaxDosVal, setKoeffProportionality := ND0603setKoefProp);
_t1033 := REAL_TO_WORD(SEL(ND0603manager.pump2ON, 0, ND0603dosing.outputValue));
ND0603regime(start := ND0603dosing.startDosingPump, pump1Main := ND0603regimeP1M, pump2Main := ND0603regimeP2M, byCounter := ND0603regimeByC, byWorkTime := ND0603regimeByWT);
ND0603manager(startStopPump1 := ND0603regime.startPump1, startStopPump2 := ND0603regime.startPump2, alarmPump1 := DD6_DI.4, alarmPump2 := DD6_DI.5, alarmReset := alarmReset, counterStart := ND0603regime.startByCounter, Pump1ResetCounter := ND0603resetCountP1, Pump2ResetCounter := ND0603resetCountP2, workTimeStart := ND0603regime.startByWorkTime, workTimePump1Reset := ND0603resetWorkTimeP1, workTimePump2Reset := ND0603resetWorkTimeP2);
ND0603dosingError := ND0603dosing.dosingError;
ND0603statRegimeP1M := ND0603regime.pump1MainActive;
ND0603statRegimeP2M := ND0603regime.pump2MainActive;
ND0603statRegimeByC := ND0603regime.byCounterActive;
ND0603statRegimeByWT := ND0603regime.byWorkTimeActive;
DD10_AO3 := _t1027;
DD10_AO4 := _t1033;
ND0603counterP1 := ND0603manager.counterPump1;
ND0603counterP2 := ND0603manager.counterPump2;
ND0603workTimeP1 := ND0603manager.currentWorkTimePump1;
ND0603workTimeP2 := ND0603manager.currentWorkTimePump2;
DD4_DO.8 := ND0603manager.pump1ON;
DD4_DO.9 := ND0603manager.pump2ON;
(* macro управление НД08.03 УПФ *)
(* сигнал 4...20мА на НД08.03/02 *)
(* сигнал 4...20мА на НД08.03/01 *)
(* Если на входе SEL = TRUE, / то нижнее значение, / иначе - то,что посередине. *)
_t1355 := SEL(ND0803manager.pump1ON, 0, ND0803dosing.outputValue);
ND0803dosing(flowValue := DD1_AI1_FT0101value, setMaxPumpDosingValue := ND0803setMaxDosVal, setKoeffProportionality := ND0803setKoefProp);
_t1361 := SEL(ND0803manager.pump2ON, 0, ND0803dosing.outputValue);
ND0803regime(start := ND0803dosing.startDosingPump, pump1Main := ND0803regimeP1M, pump2Main := ND0803regimeP2M, byCounter := ND0803regimeByC, byWorkTime := ND0803regimeByWT);
ND0803manager(startStopPump1 := ND0803regime.startPump1, startStopPump2 := ND0803regime.startPump2, alarmPump1 := DD5_DI.12 OR DD1_DI6, alarmPump2 := DD5_DI.13 OR DD1_DI7, alarmReset := alarmReset, counterStart := ND0803regime.startByCounter, Pump1ResetCounter := ND0803resetCountP1, Pump2ResetCounter := ND0803resetCountP2, workTimeStart := ND0803regime.startByWorkTime, workTimePump1Reset := ND0803resetWorkTimeP1, workTimePump2Reset := ND0803resetWorkTimeP2);
ND0803dosingError := ND0803dosing.dosingError;
ND0803statRegimeP1M := ND0803regime.pump1MainActive;
ND0803statRegimeP2M := ND0803regime.pump2MainActive;
ND0803statRegimeByC := ND0803regime.byCounterActive;
ND0803statRegimeByWT := ND0803regime.byWorkTimeActive;
DD1_AO1 := _t1355;
DD1_AO2 := _t1361;
ND0803counterP1 := ND0803manager.counterPump1;
ND0803counterP2 := ND0803manager.counterPump2;
ND0803workTimeP1 := ND0803manager.currentWorkTimePump1;
ND0803workTimeP2 := ND0803manager.currentWorkTimePump2;
DD1_DO3 := ND0803manager.pump1ON;
DD1_DO4 := ND0803manager.pump2ON;
(* macro управление НД07.03 УПЩ (поддержка рН, ПИД-регулятор) *)
(* сигнал 4...20мА на НД07.03/02 *)
(* сигнал 4...20мА на НД07.03/01 *)
(* Если на входе SEL = TRUE, / то нижнее значение, / иначе - то,что посередине. *)
(* min расход в кубометрах в час / для неачала дозирования. *)
ND0703pidReg(ACTUAL := DD1_AI3_QE0101value, SET_POINT := ND0703pHsetValue, KP := ND0703koeffP, TN := ND0703koeffI, TV := ND0703koeffD, Y_MANUAL := ND0703YoutManual, Y_OFFSET := 12, Y_MIN := 4, Y_MAX := 20, MANUAL := ND0703YmanAuto, RESET := ND0703pidReg.OVERFLOW);
_t1183 := REAL_TO_WORD(SEL(ND0703manager.pump1ON, 0, ND0703pidReg.Y));
_t1189 := REAL_TO_WORD(SEL(ND0703manager.pump2ON, 0, ND0703pidReg.Y));
ND0703regime(start := DD1_AI1_FT0101value >= 10, pump1Main := ND0703regimeP1M, pump2Main := ND0703regimeP2M, byCounter := ND0703regimeByC, byWorkTime := ND0703regimeByWT);
ND0703manager(startStopPump1 := ND0703regime.startPump1, startStopPump2 := ND0703regime.startPump2, alarmPump1 := DD6_DI.6, alarmPump2 := DD6_DI.7, alarmReset := alarmReset, counterStart := ND0703regime.startByCounter, Pump1ResetCounter := ND0703resetCountP1, Pump2ResetCounter := ND0703resetCountP2, workTimeStart := ND0703regime.startByWorkTime, workTimePump1Reset := ND0703resetWorkTimeP1, workTimePump2Reset := ND0703resetWorkTimeP2);
ND0703statRegimeP1M := ND0703regime.pump1MainActive;
ND0703statRegimeP2M := ND0703regime.pump2MainActive;
ND0703statRegimeByC := ND0703regime.byCounterActive;
ND0703statRegimeByWT := ND0703regime.byWorkTimeActive;
DD10_AO5 := _t1183;
DD10_AO6 := _t1189;
ND0703counterP1 := ND0703manager.counterPump1;
ND0703counterP2 := ND0703manager.counterPump2;
ND0703workTimeP1 := ND0703manager.currentWorkTimePump1;
ND0703workTimeP2 := ND0703manager.currentWorkTimePump2;
DD4_DO.10 := ND0703manager.pump1ON;
DD4_DO.11 := ND0703manager.pump2ON;
(* macro управление НД08.04 УПФ *)
(* Преобразует сигнал 0...100 / пропорционально в 4...20мА *)
_t1403 := DD7_DI.13 AND _t1404;
_t1404 := NOT DD6_DI.16;
ND0804linearTransformator(IN := ND0804doseValue, IN_MIN := 0, IN_MAX := 100, OUT_MIN := 4, OUT_MAX := 20);
DD4_DO.12 := _t1403;
DD10_AO7 := REAL_TO_WORD(ND0804linearTransformator.OUT);
ND0804dosingError := ND0804linearTransformator.ERROR;
(* macro контроль температуры в помещении *)
(* задаем границы допустимой температуры в помещении / проверяем что измеренное значение в заданном диапазоне *)
(* не смотрим конкретный тип ошибки / (работает не точно, обрыв определяет как слишком маленькое значение) / если не равно 0 - значит на входе ошибка *)
DD1_AI0_temperature(VALUE := DD1_AI0);
temperatureLimits(IN := REAL_TO_INT(DD1_AI0_temperature.OUT_VALUE), HIGH := minTemperature, LOW := maxTemperature);
temperatureLimits();
temperatureValue := DD1_AI0_temperature.OUT_VALUE;
DD1_AI0_error := DD1_AI0_temperature._ERR <> 0;
alarmHighTemperature := temperatureLimits.O;
alarmLowTemperature := temperatureLimits.U;
tempTwoPumpOneDriveManager(startStopPump1 := temp1, startStopPump2 := temp2, alarmPump1 := temp3, alarmPump2 := temp4, alarmReset := temp5, counterStart := temp6, Pump1ResetCounter := temp7, Pump2ResetCounter := temp8, workTimeStart := temp9, workTimePump1Reset := temp10, workTimePump2Reset := temp11);
temp12 := tempTwoPumpOneDriveManager.counterPump1;
temp13 := tempTwoPumpOneDriveManager.counterPump2;
temp14 := tempTwoPumpOneDriveManager.currentWorkTimePump1;
temp15 := tempTwoPumpOneDriveManager.currentWorkTimePump2;
temp16 := tempTwoPumpOneDriveManager.DriveKM;
temp17 := tempTwoPumpOneDriveManager.pump1KM;
temp18 := tempTwoPumpOneDriveManager.pump2KM;
temp19 := tempTwoPumpOneDriveManager.driveStart;
END_PROGRAM

(* POU DosingPumpProportional, CFC *)
FUNCTION_BLOCK DosingPumpProportional
VAR_INPUT
	flowValue: REAL;		(*текущее значение мгновенного расхода, кубометров в час.*)
	setMinPumpDosingValue: REAL := 0;		(*задание минимальной производительности доз.насоса.
По умолчанию, если ничего не подключено ко входу, равно нулю.*)
	setMaxPumpDosingValue: REAL;		(*задание максимальной производительности доз.насоса, в мл/мин*)
	minOutputValue: REAL := 4;		(*минимальное значение выходного сигнала.
По умолчанию, если ничего не подключено ко входу, равно 4.*)
	maxOutputValue: REAL := 20;		(*Максимально значение выходного сигнала.
			По умолчанию, если ничего не подключено ко входу, равно 20.*)
	setKoeffProportionality: REAL;		(*Задание мл на кубометр (коэф.пропорциональности между расходом и дозированием)*)
	minFlowToStart: REAL := 10;		(*Минимальное значение расхода для подачи сигнала на начало дозирования.
			По умолчанию, если ничего не подключено ко входу, равно 10 кубометров в час.*)
END_VAR
VAR_OUTPUT
	outputValue: REAL;		(*Выходной сигнал на дозирующий насос.*)
	dosingError: BOOL;		(*Ошибка производительности дозирования (неверно заданы значения производительности насоса, производительность доз.насоса не соответствует расходу.*)
	startDosingPump: BOOL;		(*Сигнал на запуск дозирующего насоса.*)
END_VAR
VAR
	linearTransformator: LIN_TRAFO;		(*получает на вход значение из указанного диапазона, ставит на выходе пропорциональное значение из другого диапазона.*)
END_VAR
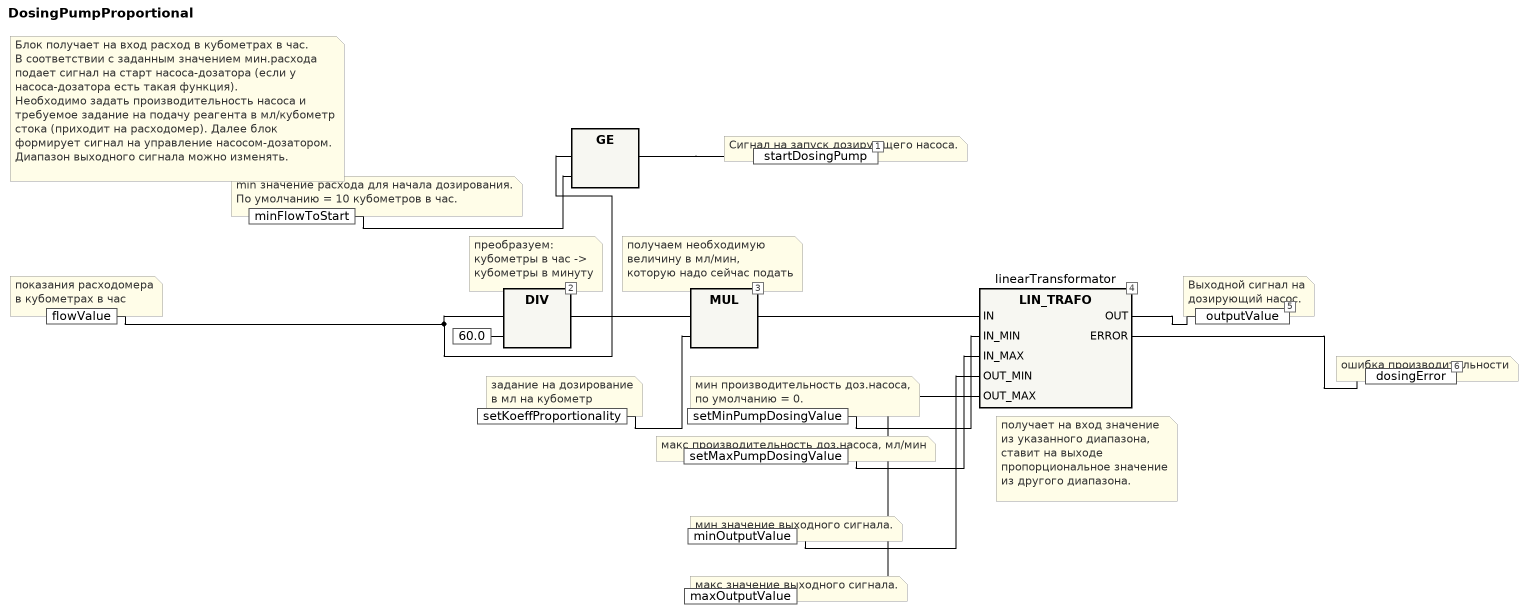
_CFC_ (* Continuous Function Chart, elements in execution order *)
(* Сигнал на запуск дозирующего насоса. *)
(* min значение расхода для начала дозирования. / По умолчанию = 10 кубометров в час. *)
(* макс производительность доз.насоса, мл/мин *)
(* мин производительность доз.насоса, / по умолчанию = 0. *)
(* получаем необходимую / величину в мл/мин, / которую надо сейчас подать *)
(* задание на дозирование / в мл на кубометр *)
(* показания расходомера / в кубометрах в час *)
(* преобразуем: / кубометры в час -> / кубометры в минуту *)
(* мин значение выходного сигнала. *)
(* макс значение выходного сигнала. *)
(* Выходной сигнал на / дозирующий насос. *)
(* ошибка производительности *)
(* получает на вход значение / из указанного диапазона, / ставит на выходе / пропорциональное значение / из другого диапазона. *)
(* Блок получает на вход расход в кубометрах в час. / В соответствии с заданным значением мин.расхода подает сигнал на старт насоса-дозатора (если у насоса-дозатора есть такая функция). / Необходимо задать производительность насоса и требуемое задание на подачу реагента в мл/кубометр стока (приходит на расходомер). Далее блок формирует сигнал на управление насосом-дозатором. / Диапазон выходного сигнала можно изменять. *)
#0 GE(flowValue, minFlowToStart)
#1 startDosingPump <= #0
#2 DIV(flowValue, 60.0)
#3 MUL(#2, setKoeffProportionality)
#4 linearTransformator:LIN_TRAFO(IN: #3, IN_MIN: setMinPumpDosingValue, IN_MAX: setMaxPumpDosingValue, OUT_MIN: minOutputValue, OUT_MAX: maxOutputValue)
#5 outputValue <= #4.OUT
#6 dosingError <= #4.ERROR
_END_CFC_
(* the same logic as Structured Text *)
(* Сигнал на запуск дозирующего насоса. *)
(* min значение расхода для начала дозирования. / По умолчанию = 10 кубометров в час. *)
(* макс производительность доз.насоса, мл/мин *)
(* мин производительность доз.насоса, / по умолчанию = 0. *)
(* получаем необходимую / величину в мл/мин, / которую надо сейчас подать *)
(* задание на дозирование / в мл на кубометр *)
(* показания расходомера / в кубометрах в час *)
(* преобразуем: / кубометры в час -> / кубометры в минуту *)
(* мин значение выходного сигнала. *)
(* макс значение выходного сигнала. *)
(* Выходной сигнал на / дозирующий насос. *)
(* ошибка производительности *)
(* получает на вход значение / из указанного диапазона, / ставит на выходе / пропорциональное значение / из другого диапазона. *)
(* Блок получает на вход расход в кубометрах в час. / В соответствии с заданным значением мин.расхода подает сигнал на старт насоса-дозатора (если у насоса-дозатора есть такая функция). / Необходимо задать производительность насоса и требуемое задание на подачу реагента в мл/кубометр стока (приходит на расходомер). Далее блок формирует сигнал на управление насосом-дозатором. / Диапазон выходного сигнала можно изменять. *)
startDosingPump := flowValue >= minFlowToStart;
linearTransformator(IN := (flowValue / 60.0) * setKoeffProportionality, IN_MIN := setMinPumpDosingValue, IN_MAX := setMaxPumpDosingValue, OUT_MIN := minOutputValue, OUT_MAX := maxOutputValue);
outputValue := linearTransformator.OUT;
dosingError := linearTransformator.ERROR;
END_FUNCTION_BLOCK

(* POU choosePumpRegime, CFC *)
FUNCTION_BLOCK choosePumpRegime
VAR
	pump1RStrig: RS;		(*Триггер-защелка выбора режима с главным первым насосом.*)
	pump2RStrig: RS;		(*Триггер-защелка выбора режима с главным вторым насосом.*)
	byCounterRStrig: RS;		(*Триггер-защелка выбора режима с запуском по количеству включений.*)
	byWorkTimeRStrig: RS;		(*Триггер-защелка выбора режима с запуском по наработке.*)
	Pump1MainDetector: R_TRIG;		(*Детектор переднего фронта включения режима, когда главный насос - первый.
			Для сброса остальных значений.*)
	Pump2MainDetector: R_TRIG;		(*Детектор переднего фронта включения режима, когда главный насос - второй.
			Для сброса остальных значений.*)
	ByCounterDetector: R_TRIG;		(*Детектор переднего фронта включения режима по количеству включений.
			Для сброса остальных значений.*)
	ByWorkTimeDetector: R_TRIG;		(*Детектор переднего фронта включения режима по наработке.
			Для сброса остальных значений.*)
END_VAR
VAR_INPUT
	start: BOOL;		(*Сигнал на включение насоса.
			Активируется выход согласно выбранного режима.*)
	pump1Main: BOOL;		(*Режим: первый насос главный, второй - резервный.*)
	pump2Main: BOOL;		(*Режим: второй насос главный, первый - резервный.*)
	byCounter: BOOL;		(*Режим: запуск по количеству включений.
			Включится с меньшим количеством стартов.*)
	byWorkTime: BOOL;		(*Режим: запуск по наработке.
			Включится насос с меньшей наработкой.*)
END_VAR
VAR_OUTPUT
	pump1MainActive: BOOL;		(*Активный режим: первый насос главный.*)
	pump2MainActive: BOOL;		(*Активный режим: второй насос главный.*)
	byCounterActive: BOOL;		(*Активный режим: включение по количеству запусков.*)
	byWorkTimeActive: BOOL;		(*Активный режим: по наработке.*)
	startPump1: BOOL;		(*Запуск первого насоса как главного (основного).*)
	startPump2: BOOL;		(*Запуск второго насоса как главного (основного).*)
	startByCounter: BOOL;		(*Запуск насоса по количеству стартов.
			Запустится с меньшим. Если одинаково, то - первый.*)
	startByWorkTime: BOOL;		(*Запуск по наработке.
			Включится с меньшей. Если одинаково, то - первый.*)
END_VAR
VAR (* helpers for the ST form of the networks *)
	_en62 : BOOL;
	_t62 : BOOL;
	_en72 : BOOL;
	_t72 : BOOL;
	_en78 : BOOL;
	_t78 : BOOL;
	_en84 : BOOL;
	_t84 : BOOL;
END_VAR
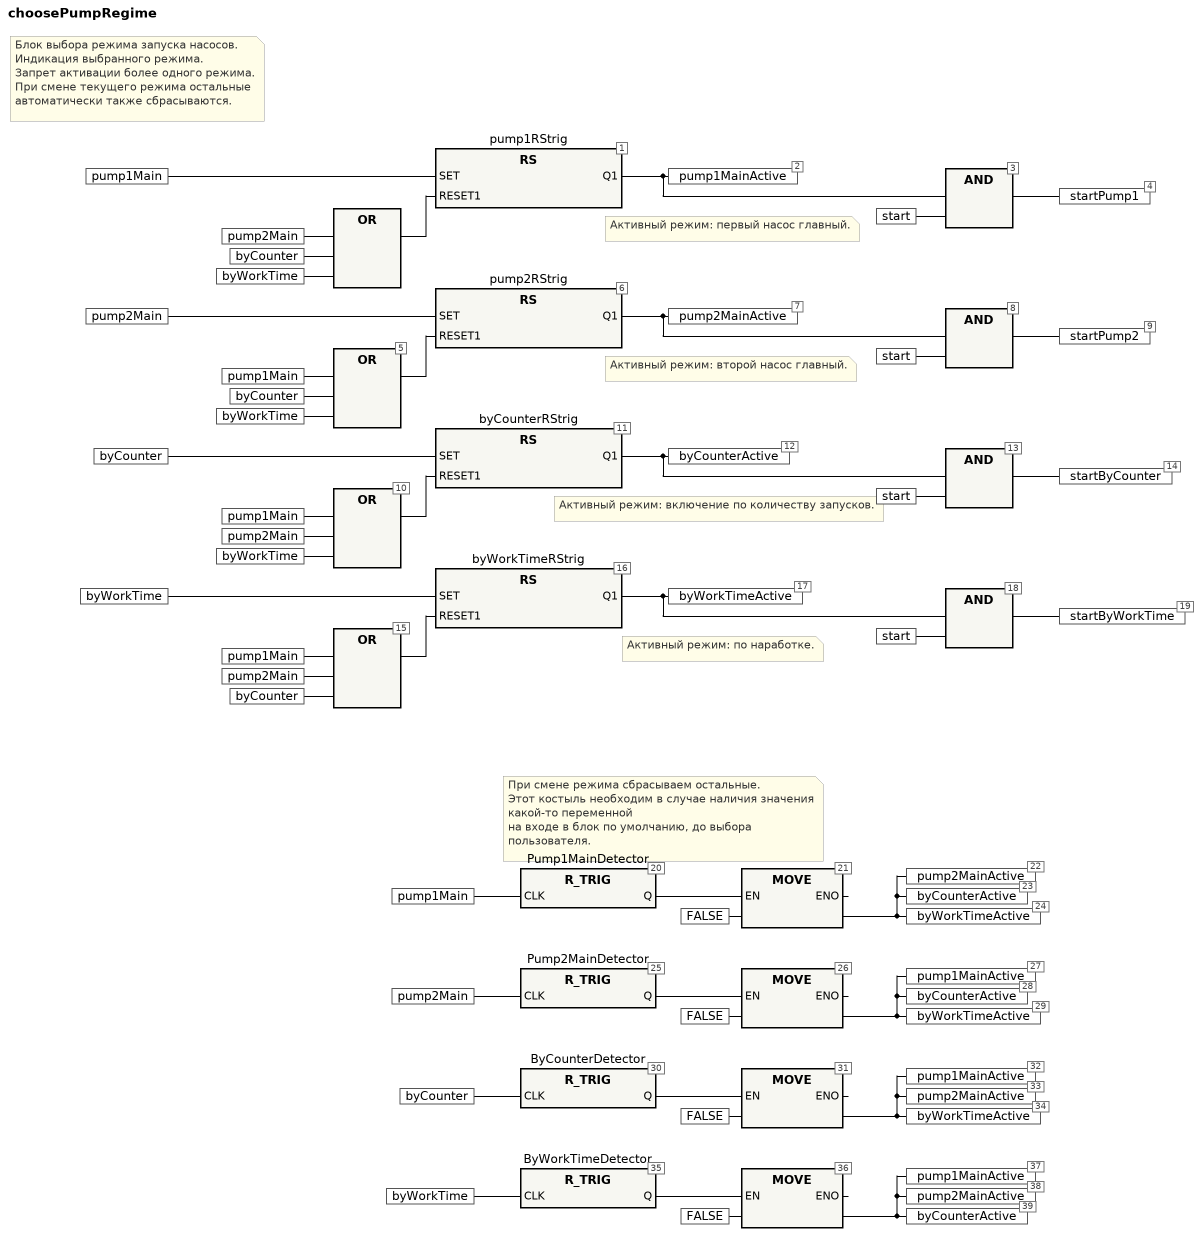
_CFC_ (* Continuous Function Chart, elements in execution order *)
(* Блок выбора режима запуска насосов. / Индикация выбранного режима. / Запрет активации более одного режима. / При смене текущего режима остальные автоматически также сбрасываются. *)
(* Активный режим: первый насос главный. *)
(* Активный режим: включение по количеству запусков. *)
(* Активный режим: по наработке. *)
(* Активный режим: второй насос главный. *)
(* При смене режима сбрасываем остальные. / Этот костыль необходим в случае наличия значения какой-то переменной / на входе в блок по умолчанию, до выбора пользователя. *)
#0 OR(pump2Main, byCounter, byWorkTime)
#1 pump1RStrig:RS(SET: pump1Main, RESET1: #0)
#2 pump1MainActive <= #1.Q1
#3 AND(#1.Q1, start)
#4 startPump1 <= #3
#5 OR(pump1Main, byCounter, byWorkTime)
#6 pump2RStrig:RS(SET: pump2Main, RESET1: #5)
#7 pump2MainActive <= #6.Q1
#8 AND(#6.Q1, start)
#9 startPump2 <= #8
#10 OR(pump1Main, pump2Main, byWorkTime)
#11 byCounterRStrig:RS(SET: byCounter, RESET1: #10)
#12 byCounterActive <= #11.Q1
#13 AND(#11.Q1, start)
#14 startByCounter <= #13
#15 OR(pump1Main, pump2Main, byCounter)
#16 byWorkTimeRStrig:RS(SET: byWorkTime, RESET1: #15)
#17 byWorkTimeActive <= #16.Q1
#18 AND(#16.Q1, start)
#19 startByWorkTime <= #18
#20 Pump1MainDetector:R_TRIG(CLK: pump1Main)
#21 MOVE(EN: #20.Q, FALSE)
#22 pump2MainActive <= #21
#23 byCounterActive <= #21
#24 byWorkTimeActive <= #21
#25 Pump2MainDetector:R_TRIG(CLK: pump2Main)
#26 MOVE(EN: #25.Q, FALSE)
#27 pump1MainActive <= #26
#28 byCounterActive <= #26
#29 byWorkTimeActive <= #26
#30 ByCounterDetector:R_TRIG(CLK: byCounter)
#31 MOVE(EN: #30.Q, FALSE)
#32 pump1MainActive <= #31
#33 pump2MainActive <= #31
#34 byWorkTimeActive <= #31
#35 ByWorkTimeDetector:R_TRIG(CLK: byWorkTime)
#36 MOVE(EN: #35.Q, FALSE)
#37 pump1MainActive <= #36
#38 pump2MainActive <= #36
#39 byCounterActive <= #36
_END_CFC_
(* the same logic as Structured Text *)
(* Блок выбора режима запуска насосов. / Индикация выбранного режима. / Запрет активации более одного режима. / При смене текущего режима остальные автоматически также сбрасываются. *)
(* Активный режим: первый насос главный. *)
(* Активный режим: включение по количеству запусков. *)
(* Активный режим: по наработке. *)
(* Активный режим: второй насос главный. *)
(* При смене режима сбрасываем остальные. / Этот костыль необходим в случае наличия значения какой-то переменной / на входе в блок по умолчанию, до выбора пользователя. *)
pump1RStrig(SET := pump1Main, RESET1 := pump2Main OR byCounter OR byWorkTime);
pump1MainActive := pump1RStrig.Q1;
startPump1 := pump1RStrig.Q1 AND start;
pump2RStrig(SET := pump2Main, RESET1 := pump1Main OR byCounter OR byWorkTime);
pump2MainActive := pump2RStrig.Q1;
startPump2 := pump2RStrig.Q1 AND start;
byCounterRStrig(SET := byCounter, RESET1 := pump1Main OR pump2Main OR byWorkTime);
byCounterActive := byCounterRStrig.Q1;
startByCounter := byCounterRStrig.Q1 AND start;
byWorkTimeRStrig(SET := byWorkTime, RESET1 := pump1Main OR pump2Main OR byCounter);
byWorkTimeActive := byWorkTimeRStrig.Q1;
startByWorkTime := byWorkTimeRStrig.Q1 AND start;
Pump1MainDetector(CLK := pump1Main);
_en62 := Pump1MainDetector.Q;
IF _en62 THEN _t62 := FALSE; END_IF;
IF _en62 THEN pump2MainActive := _t62; END_IF;
IF _en62 THEN byCounterActive := _t62; END_IF;
IF _en62 THEN byWorkTimeActive := _t62; END_IF;
Pump2MainDetector(CLK := pump2Main);
_en72 := Pump2MainDetector.Q;
IF _en72 THEN _t72 := FALSE; END_IF;
IF _en72 THEN pump1MainActive := _t72; END_IF;
IF _en72 THEN byCounterActive := _t72; END_IF;
IF _en72 THEN byWorkTimeActive := _t72; END_IF;
ByCounterDetector(CLK := byCounter);
_en78 := ByCounterDetector.Q;
IF _en78 THEN _t78 := FALSE; END_IF;
IF _en78 THEN pump1MainActive := _t78; END_IF;
IF _en78 THEN pump2MainActive := _t78; END_IF;
IF _en78 THEN byWorkTimeActive := _t78; END_IF;
ByWorkTimeDetector(CLK := byWorkTime);
_en84 := ByWorkTimeDetector.Q;
IF _en84 THEN _t84 := FALSE; END_IF;
IF _en84 THEN pump1MainActive := _t84; END_IF;
IF _en84 THEN pump2MainActive := _t84; END_IF;
IF _en84 THEN byCounterActive := _t84; END_IF;
END_FUNCTION_BLOCK

(* POU TwoPumpManager, CFC *)
FUNCTION_BLOCK TwoPumpManager
VAR_INPUT
	startStopPump1: BOOL;		(*Сигнал на пуск/стоп первого насоса.*)
	startStopPump2: BOOL;		(*Сигнал на пуск/стоп второго насоса.*)
	alarmPump1: BOOL;		(*Сигнал "авария" на первом насосе.*)
	alarmPump2: BOOL;		(*Сигнал "авария" на втором насосе.*)
	alarmReset: BOOL;		(*Сброс аварии.*)

	counterStart: BOOL;		(*Запуск насоса с меньшим количеством включений.*)
	Pump1ResetCounter: BOOL;		(*Сброс счетчика количества включений первого насоса.
Сбрасывается также автоматически при достижении счетчиком значения ValueToResetCTU.*)
	Pump2ResetCounter: BOOL;		(*Сброс счетчика количества включений второго насоса.
Сбрасывается также автоматически при достижении счетчиком значения ValueToResetCTU.*)
	ValueToResetCounter: WORD := 32767;		(*Значение счетчика, после которого он сбрасывается на ноль.
			Максимальное допустимое значение: 32767, будет установлено, если не подключать ничего на вход.*)

	workTimeStart: BOOL;		(*Запуск насоса с выбором по меньшей наработке.*)
	workTimePump1Reset: BOOL;		(*Сброс времени наработки первого насоса.*)
	workTimePump2Reset: BOOL;		(*Сброс времени наработки второго насоса.*)
END_VAR
VAR_OUTPUT
	pump1ON: BOOL;		(*Выход на включение первого насоса.*)
	pump2ON: BOOL;		(*Выход на включение второго насоса.*)

	counterPump1: WORD;		(*Количество включений первого насоса.
При достижении значения ValueToResetCTU сбрасывается в ноль.*)
	counterPump2: WORD;		(*Количество включений второго насоса.
При достижении значения ValueToResetCTU сбрасывается в ноль.*)

	currentWorkTimePump1: TIME;		(*Текущая наработка первого насоса.*)
	currentWorkTimePump2: TIME;		(*Текущая наработка второго насоса.*)
END_VAR
VAR
	RtrigPump1: R_TRIG;		(*Включает первый насос по фронту сигнала на ручной пуск/стоп.*)
	FtrigPump1: F_TRIG;		(*Выключает первый насос по спаду сигнала на ручной пуск/стоп.*)
	RtrigPump2: R_TRIG;		(*Включает второй насос по фронту сигнала на ручной пуск/стоп.*)
	FtrigPump2: F_TRIG;		(*Выключает второй насос по спаду сигнала на ручной пуск/стоп.*)
	RSpump1: RS;		(*RS-триггер нормального включения первого насоса*)
	RSpump2: RS;		(*RS-триггер нормального включения второго насоса*)
	pump1NormalON: BOOL;		(*Сигнал нормального (неаварийного) включения первого насоса.*)
	pump2NormalON: BOOL;		(*Сигнал нормального (неаварийного) включения второго насоса.*)
	pump2EmergencyON: BOOL;		(*Сигнал аварийного включения второго насоса (при аварии первого).*)
	pump1EmergencyON: BOOL;		(*Сигнал аварийного включения первого насоса (при аварии второго).*)
	alarmPump1RStrig: RS;		(*Триггер аварии первого насоса.*)
	alarmPump2RStrig: RS;		(*Триггер аварии второго насоса.*)
	TONtoOnPump1: TON;		(*Таймер задержки включения первого насоса, на переключение контакторов при аварийном переключении.
			Жестко задано 1 секунда.*)
	TONtoOnPump2: TON;		(*Таймер задержки включения второго насоса, на переключение контакторов при аварийном переключении.
						Жестко задано 1 секунда.*)

	CTUPump1: CTU;		(*Счетчик количества включений первого насоса.*)
	CTUPump2: CTU;		(*Счетчик количества включений второго насоса.*)
	counterRtrig: R_TRIG;		(*Детектор переднего фронта сигнала на старт насоса с меньшей наработкой, включает насос.*)
	counterFtrig: F_TRIG;		(*Детектор спада сигнала на запуск насоса с меньшей наработкой, останавливает насос.*)
	counterRStrigPump1: RS;		(*Триггер-защелка включения первого насоса при запуске по количеству включений.*)
	counterRStrigPump2: RS;		(*Триггер-защелка включения второго насоса при запуске по количеству включений.*)
	counterPump1ON: BOOL;		(*Сигнал на запуск первого насоса при запуске по количеству включений.*)
	counterPump2ON: BOOL;		(*Сигнал на запуск второго насоса при запуске по количеству включений.*)

	workTimePump1ON: BOOL;		(*Сигнал на запуск первого насоса при запуске по наработке.*)
	workTimePump2ON: BOOL;		(*Сигнал на запуск второго насоса при запуске по наработке.*)
	timerFtrig: F_TRIG;		(*Детектор спада сигнала работы насосов для записи времени работы.*)
	pump1Ftrig: F_TRIG;		(*Детектор спада сигнала работы первого насоса для подсчета наработки.*)
	pump2Ftrig: F_TRIG;		(*Детектор спада сигнала работы второго насоса для подсчета наработки.*)
	timeStartFtrig: F_TRIG;		(*Детектор спада сигнала на запуск по наработке.*)
	timeStartRtrig: R_TRIG;		(*Детектор переднего фронта сигнала на запуск по наработке.*)
	timerRTC: RTC;		(*Таймер реального времени для подсчета наработки.*)
	timeCDT: DT;		(*Время на выходе таймера реального времени.*)
	timePDT: DT;		(*Время на входе таймера реального времени. Не инициализируется, чтобы подсчет всегда начинался от нуля.*)
	tempVarTime: TIME;		(*Промежуточная переменная хранения времени наработки за включение.*)
	workTimePump1: TIME;		(*Время наработки первого насоса. Подсчитывается после выключения насоса.*)
	workTimePump2: TIME;		(*Время наработки второго насоса. Подсчитывается после выключения насоса.*)
	RStrigTimePump1: RS;		(*Триггер-защелка запуск первого насоса по наработке.*)
	RStrigTimePump2: RS;		(*Триггер-защелка запуск второго насоса по наработке.*)

END_VAR
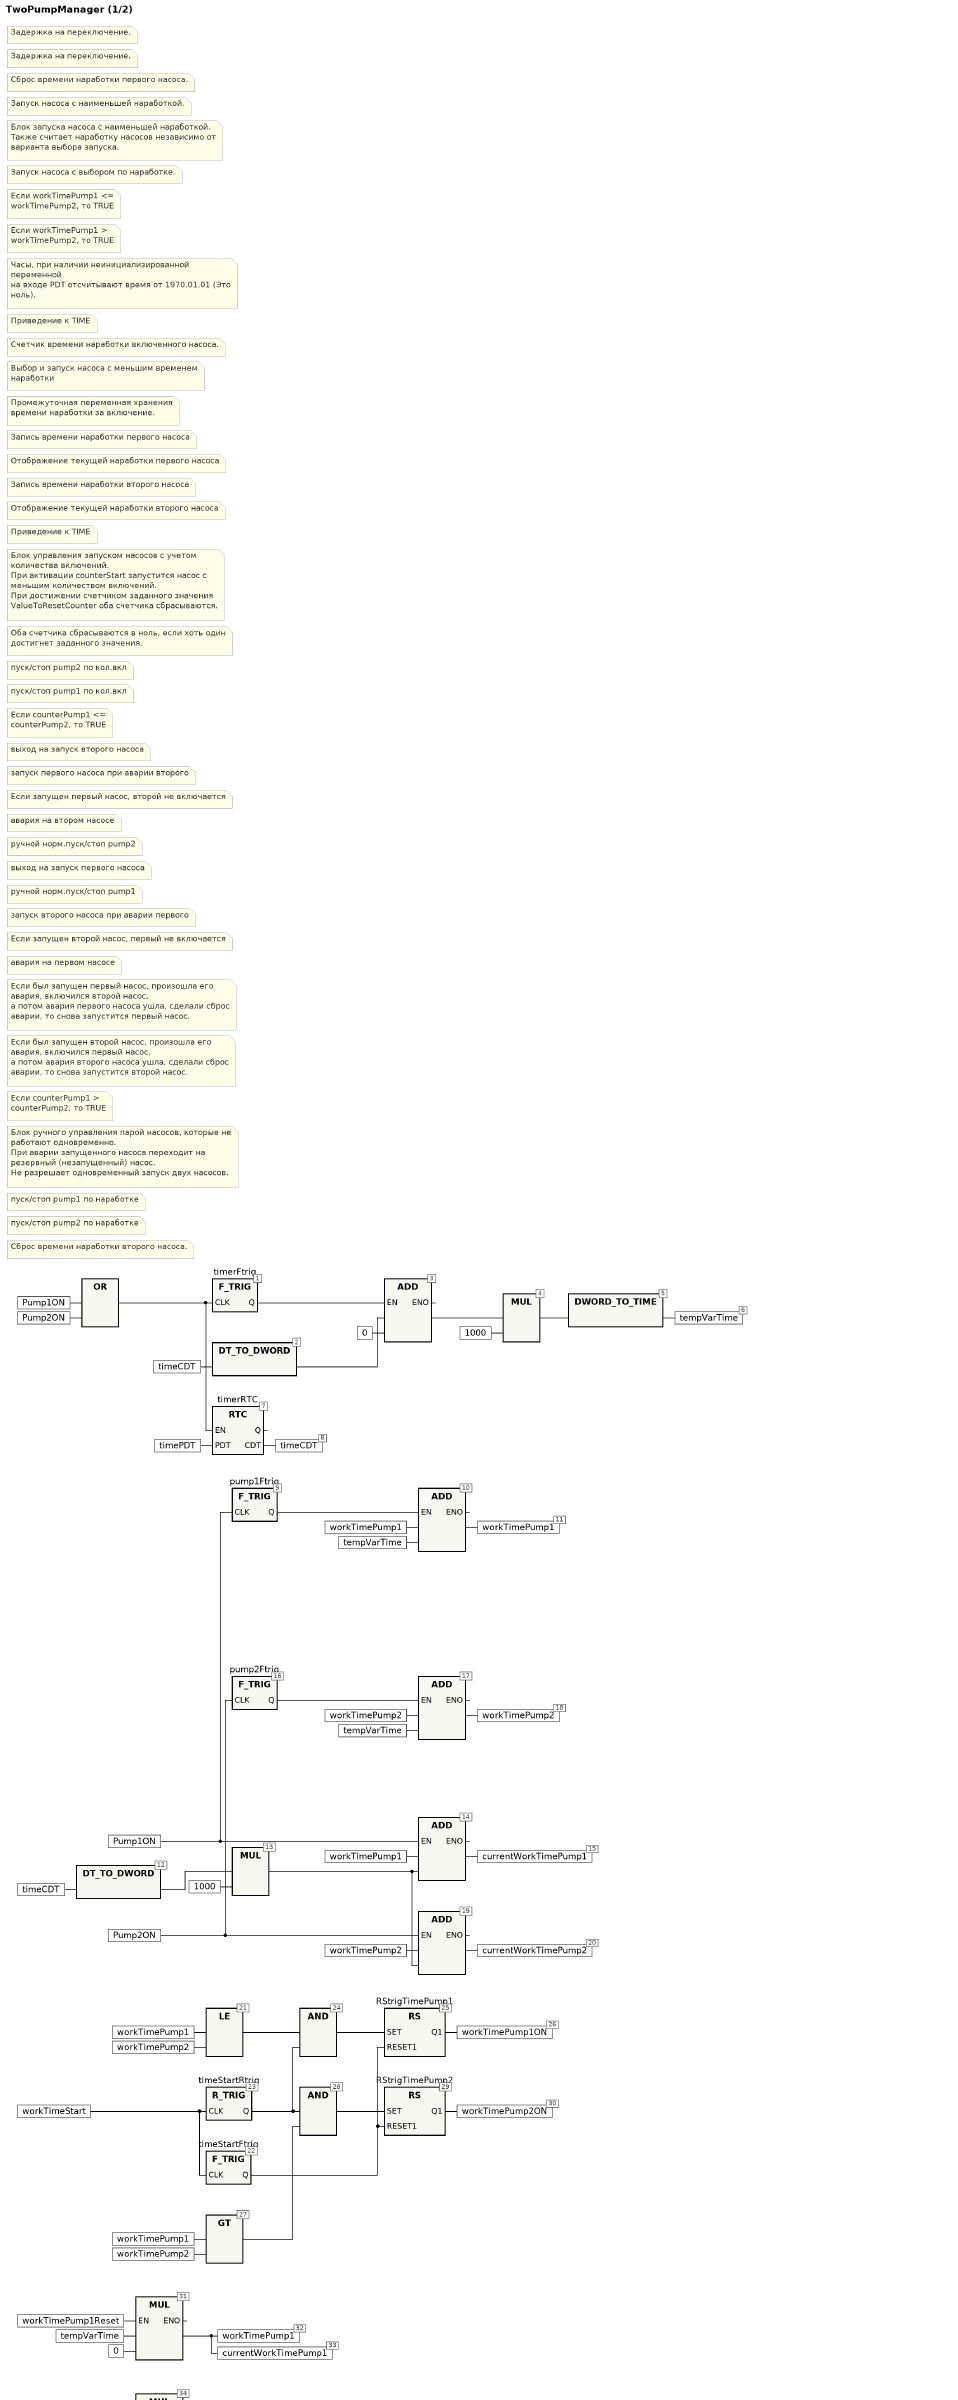
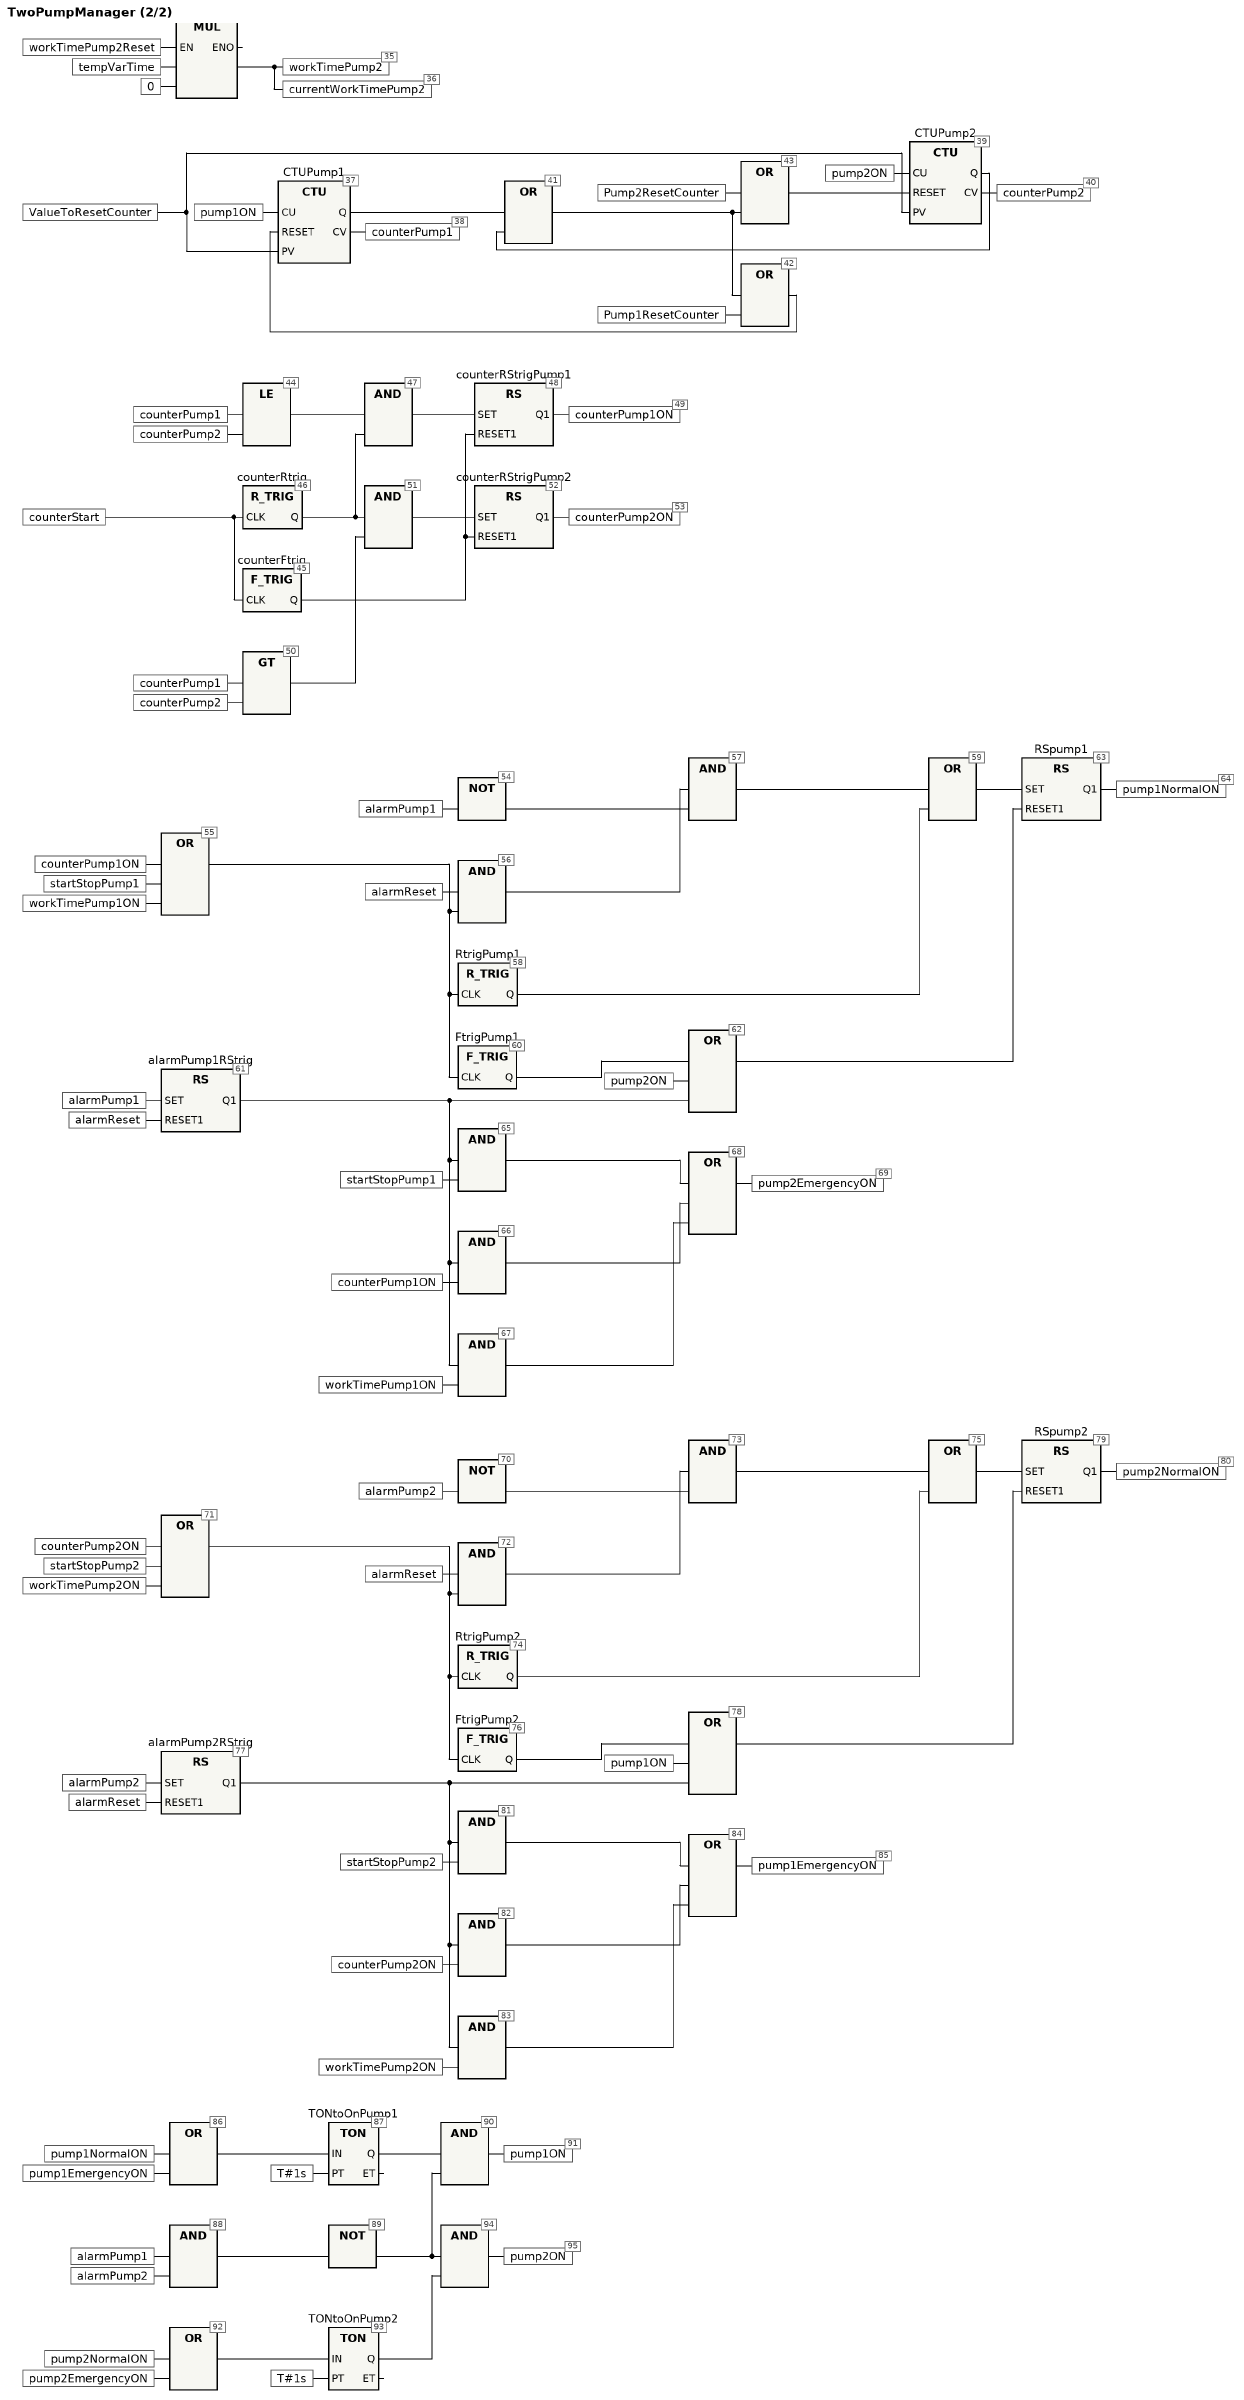
_CFC_ (* Continuous Function Chart, elements in execution order *)
(* Задержка на переключение. *)
(* Задержка на переключение. *)
(* Сброс времени наработки первого насоса. *)
(* Запуск насоса с наименьшей наработкой. *)
(* Блок запуска насоса с наименьшей наработкой. / Также считает наработку насосов независимо от варианта выбора запуска. *)
(* Запуск насоса с выбором по наработке. *)
(* Если workTimePump1 <= / workTimePump2, то TRUE *)
(* Если workTimePump1 > / workTimePump2, то TRUE *)
(* Часы, при наличии неинициализированной переменной / на входе PDT отсчитывают время от 1970.01.01 (Это ноль). *)
(* Приведение к TIME *)
(* Счетчик времени наработки включенного насоса. *)
(* Выбор и запуск насоса с меньшим временем наработки *)
(* Промежуточная переменная хранения / времени наработки за включение. *)
(* Запись времени наработки первого насоса *)
(* Отображение текущей наработки первого насоса *)
(* Запись времени наработки второго насоса *)
(* Отображение текущей наработки второго насоса *)
(* Приведение к TIME *)
(* Блок управления запуском насосов с учетом количества включений. / При активации counterStart запустится насос с меньшим количеством включений. / При достижении счетчиком заданного значения ValueToResetCounter оба счетчика сбрасываются. *)
(* Оба счетчика сбрасываются в ноль, если хоть один достигнет заданного значения. *)
(* пуск/стоп pump2 по кол.вкл *)
(* пуск/стоп pump1 по кол.вкл *)
(* Если counterPump1 <= / counterPump2, то TRUE *)
(* выход на запуск второго насоса *)
(* запуск первого насоса при аварии второго *)
(* Если запущен первый насос, второй не включается *)
(* авария на втором насосе *)
(* ручной норм.пуск/стоп pump2 *)
(* выход на запуск первого насоса *)
(* ручной норм.пуск/стоп pump1 *)
(* запуск второго насоса при аварии первого *)
(* Если запущен второй насос, первый не включается *)
(* авария на первом насосе *)
(* Если был запущен первый насос, произошла его авария, включился второй насос, / а потом авария первого насоса ушла, сделали сброс аварии, то снова запустится первый насос. *)
(* Если был запущен второй насос, произошла его авария, включился первый насос, / а потом авария второго насоса ушла, сделали сброс аварии, то снова запустится второй насос. *)
(* Если counterPump1 > / counterPump2, то TRUE *)
(* Блок ручного управления парой насосов, которые не работают одновременно. / При аварии запущенного насоса переходит на резервный (незапущенный) насос. / Не разрешает одновременный запуск двух насосов. *)
(* пуск/стоп pump1 по наработке *)
(* пуск/стоп pump2 по наработке *)
(* Сброс времени наработки второго насоса. *)
#0 OR(Pump1ON, Pump2ON)
#1 timerFtrig:F_TRIG(CLK: #0)
#2 DT_TO_DWORD(timeCDT)
#3 ADD(EN: #1.Q, #2, 0)
#4 MUL(#3, 1000)
#5 DWORD_TO_TIME(#4)
#6 tempVarTime <= #5
#7 timerRTC:RTC(EN: #0, PDT: timePDT)
#8 timeCDT <= #7.CDT
#9 pump1Ftrig:F_TRIG(CLK: Pump1ON)
#10 ADD(EN: #9.Q, workTimePump1, tempVarTime)
#11 workTimePump1 <= #10
#12 DT_TO_DWORD(timeCDT)
#13 MUL(#12, 1000)
#14 ADD(EN: Pump1ON, workTimePump1, #13)
#15 currentWorkTimePump1 <= #14
#16 pump2Ftrig:F_TRIG(CLK: Pump2ON)
#17 ADD(EN: #16.Q, workTimePump2, tempVarTime)
#18 workTimePump2 <= #17
#19 ADD(EN: Pump2ON, workTimePump2, #13)
#20 currentWorkTimePump2 <= #19
#21 LE(workTimePump1, workTimePump2)
#22 timeStartFtrig:F_TRIG(CLK: workTimeStart)
#23 timeStartRtrig:R_TRIG(CLK: workTimeStart)
#24 AND(#21, #23.Q)
#25 RStrigTimePump1:RS(SET: #24, RESET1: #22.Q)
#26 workTimePump1ON <= #25.Q1
#27 GT(workTimePump1, workTimePump2)
#28 AND(#23.Q, #27)
#29 RStrigTimePump2:RS(SET: #28, RESET1: #22.Q)
#30 workTimePump2ON <= #29.Q1
#31 MUL(EN: workTimePump1Reset, tempVarTime, 0)
#32 workTimePump1 <= #31
#33 currentWorkTimePump1 <= #31
#34 MUL(EN: workTimePump2Reset, tempVarTime, 0)
#35 workTimePump2 <= #34
#36 currentWorkTimePump2 <= #34
#37 CTUPump1:CTU(CU: pump1ON, RESET: #42, PV: ValueToResetCounter)
#38 counterPump1 <= #37.CV
#39 CTUPump2:CTU(CU: pump2ON, RESET: #43, PV: ValueToResetCounter)
#40 counterPump2 <= #39.CV
#41 OR(#37.Q, #39.Q)
#42 OR(#41, Pump1ResetCounter)
#43 OR(Pump2ResetCounter, #41)
#44 LE(counterPump1, counterPump2)
#45 counterFtrig:F_TRIG(CLK: counterStart)
#46 counterRtrig:R_TRIG(CLK: counterStart)
#47 AND(#44, #46.Q)
#48 counterRStrigPump1:RS(SET: #47, RESET1: #45.Q)
#49 counterPump1ON <= #48.Q1
#50 GT(counterPump1, counterPump2)
#51 AND(#46.Q, #50)
#52 counterRStrigPump2:RS(SET: #51, RESET1: #45.Q)
#53 counterPump2ON <= #52.Q1
#54 NOT(alarmPump1)
#55 OR(counterPump1ON, startStopPump1, workTimePump1ON)
#56 AND(alarmReset, #55)
#57 AND(#56, #54)
#58 RtrigPump1:R_TRIG(CLK: #55)
#59 OR(#57, #58.Q)
#60 FtrigPump1:F_TRIG(CLK: #55)
#61 alarmPump1RStrig:RS(SET: alarmPump1, RESET1: alarmReset)
#62 OR(#60.Q, pump2ON, #61.Q1)
#63 RSpump1:RS(SET: #59, RESET1: #62)
#64 pump1NormalON <= #63.Q1
#65 AND(#61.Q1, startStopPump1)
#66 AND(#61.Q1, counterPump1ON)
#67 AND(#61.Q1, workTimePump1ON)
#68 OR(#65, #66, #67)
#69 pump2EmergencyON <= #68
#70 NOT(alarmPump2)
#71 OR(counterPump2ON, startStopPump2, workTimePump2ON)
#72 AND(alarmReset, #71)
#73 AND(#72, #70)
#74 RtrigPump2:R_TRIG(CLK: #71)
#75 OR(#73, #74.Q)
#76 FtrigPump2:F_TRIG(CLK: #71)
#77 alarmPump2RStrig:RS(SET: alarmPump2, RESET1: alarmReset)
#78 OR(#76.Q, pump1ON, #77.Q1)
#79 RSpump2:RS(SET: #75, RESET1: #78)
#80 pump2NormalON <= #79.Q1
#81 AND(#77.Q1, startStopPump2)
#82 AND(#77.Q1, counterPump2ON)
#83 AND(#77.Q1, workTimePump2ON)
#84 OR(#81, #82, #83)
#85 pump1EmergencyON <= #84
#86 OR(pump1NormalON, pump1EmergencyON)
#87 TONtoOnPump1:TON(IN: #86, PT: T#1s)
#88 AND(alarmPump1, alarmPump2)
#89 NOT(#88)
#90 AND(#87.Q, #89)
#91 pump1ON <= #90
#92 OR(pump2NormalON, pump2EmergencyON)
#93 TONtoOnPump2:TON(IN: #92, PT: T#1s)
#94 AND(#89, #93.Q)
#95 pump2ON <= #94
_END_CFC_
END_FUNCTION_BLOCK

(* POU TwoPumpOneDriveManager, CFC *)
FUNCTION_BLOCK TwoPumpOneDriveManager
VAR_INPUT
	startStopPump1: BOOL;		(*Сигнал на пуск/стоп первого насоса.*)
	startStopPump2: BOOL;		(*Сигнал на пуск/стоп второго насоса.*)
	alarmPump1: BOOL;		(*Сигнал "авария" на первом насосе.*)
	alarmPump2: BOOL;		(*Сигнал "авария" на втором насосе.*)
	alarmReset: BOOL;		(*Сброс аварии.*)

	counterStart: BOOL;		(*Запуск насоса с меньшим количеством включений.*)
	Pump1ResetCounter: BOOL;		(*Сброс счетчика количества включений первого насоса.
Сбрасывается также автоматически при достижении счетчиком значения ValueToResetCTU.*)
	Pump2ResetCounter: BOOL;		(*Сброс счетчика количества включений второго насоса.
Сбрасывается также автоматически при достижении счетчиком значения ValueToResetCTU.*)
	ValueToResetCounter: WORD := 32767;		(*Значение счетчика, после которого он сбрасывается на ноль.
			Максимальное допустимое значение: 32767, будет установлено, если не подключать ничего на вход.*)

	workTimeStart: BOOL;		(*Запуск насоса с выбором по меньшей наработке.*)
	workTimePump1Reset: BOOL;		(*Сброс времени наработки первого насоса.*)
	workTimePump2Reset: BOOL;		(*Сброс времени наработки второго насоса.*)
	timeKM1off: TIME := T#20s;		(*Время на которое отключается питание ЧРП.
			По умолчанию = 20сек.*)
	timeKM23DelayON: TIME := T#15s;		(*Время задержки включения контактора насоса.
			По умолчанию = 15 сек.*)
	timeKM23offDelay: TIME := T#10s;		(*Время задержки выключения контактора насосов.
			По умолчанию = 10сек. (Чтобы сначала отключилось питание ЧРП).*)
	timeReadyToStartDelay: TIME := T#5s;		(*Время задержки подачи сигнала на старт ЧРП.
			По умолчанию = 5сек.*)
END_VAR
VAR_OUTPUT

	counterPump1: WORD;		(*Количество включений первого насоса.
При достижении значения ValueToResetCTU сбрасывается в ноль.*)
	counterPump2: WORD;		(*Количество включений второго насоса.
При достижении значения ValueToResetCTU сбрасывается в ноль.*)

	currentWorkTimePump1: TIME;		(*Текущая наработка первого насоса.*)
	currentWorkTimePump2: TIME;		(*Текущая наработка второго насоса.*)

	DriveKM: BOOL;		(*Выход на включение контактора частотного преобразователя (питание).*)
	pump1KM: BOOL;		(*Выход на включение контактора первого насоса.*)
	pump2KM: BOOL;		(*Выход на включение контактора второго насоса.*)
	driveStart: BOOL;		(*Сигнал на старт частотного преобразователя.*)
END_VAR
VAR
	RtrigPump1: R_TRIG;		(*Включает первый насос по фронту сигнала на ручной пуск/стоп.*)
	FtrigPump1: F_TRIG;		(*Выключает первый насос по спаду сигнала на ручной пуск/стоп.*)
	RtrigPump2: R_TRIG;		(*Включает второй насос по фронту сигнала на ручной пуск/стоп.*)
	FtrigPump2: F_TRIG;		(*Выключает второй насос по спаду сигнала на ручной пуск/стоп.*)
	RSpump1: RS;		(*RS-триггер нормального включения первого насоса*)
	RSpump2: RS;		(*RS-триггер нормального включения второго насоса*)
	pump1NormalON: BOOL;		(*Сигнал нормального (неаварийного) включения первого насоса.*)
	pump2NormalON: BOOL;		(*Сигнал нормального (неаварийного) включения второго насоса.*)
	pump2EmergencyON: BOOL;		(*Сигнал аварийного включения второго насоса (при аварии первого).*)
	pump1EmergencyON: BOOL;		(*Сигнал аварийного включения первого насоса (при аварии второго).*)
	alarmPump1RStrig: RS;		(*Триггер аварии первого насоса.*)
	alarmPump2RStrig: RS;		(*Триггер аварии второго насоса.*)
	TONtoOnPump1: TON;		(*Таймер задержки включения первого насоса, на переключение контакторов при аварийном переключении.
			Жестко задано 1 секунда.*)
	TONtoOnPump2: TON;		(*Таймер задержки включения второго насоса, на переключение контакторов при аварийном переключении.
						Жестко задано 1 секунда.*)

	CTUPump1: CTU;		(*Счетчик количества включений первого насоса.*)
	CTUPump2: CTU;		(*Счетчик количества включений второго насоса.*)
	counterRtrig: R_TRIG;		(*Детектор переднего фронта сигнала на старт насоса с меньшей наработкой, включает насос.*)
	counterFtrig: F_TRIG;		(*Детектор спада сигнала на запуск насоса с меньшей наработкой, останавливает насос.*)
	counterRStrigPump1: RS;		(*Триггер-защелка включения первого насоса при запуске по количеству включений.*)
	counterRStrigPump2: RS;		(*Триггер-защелка включения второго насоса при запуске по количеству включений.*)
	counterPump1ON: BOOL;		(*Сигнал на запуск первого насоса при запуске по количеству включений.*)
	counterPump2ON: BOOL;		(*Сигнал на запуск второго насоса при запуске по количеству включений.*)

	workTimePump1ON: BOOL;		(*Сигнал на запуск первого насоса при запуске по наработке.*)
	workTimePump2ON: BOOL;		(*Сигнал на запуск второго насоса при запуске по наработке.*)
	timerFtrig: F_TRIG;		(*Детектор спада сигнала работы насосов для записи времени работы.*)
	pump1Ftrig: F_TRIG;		(*Детектор спада сигнала работы первого насоса для подсчета наработки.*)
	pump2Ftrig: F_TRIG;		(*Детектор спада сигнала работы второго насоса для подсчета наработки.*)
	timeStartFtrig: F_TRIG;		(*Детектор спада сигнала на запуск по наработке.*)
	timeStartRtrig: R_TRIG;		(*Детектор переднего фронта сигнала на запуск по наработке.*)
	timerRTC: RTC;		(*Таймер реального времени для подсчета наработки.*)
	timeCDT: DT;		(*Время на выходе таймера реального времени.*)
	timePDT: DT;		(*Время на входе таймера реального времени. Не инициализируется, чтобы подсчет всегда начинался от нуля.*)
	tempVarTime: TIME;		(*Промежуточная переменная хранения времени наработки за включение.*)
	workTimePump1: TIME;		(*Время наработки первого насоса. Подсчитывается после выключения насоса.*)
	workTimePump2: TIME;		(*Время наработки второго насоса. Подсчитывается после выключения насоса.*)
	RStrigTimePump1: RS;		(*Триггер-защелка запуск первого насоса по наработке.*)
	RStrigTimePump2: RS;		(*Триггер-защелка запуск второго насоса по наработке.*)

	pump1ON: BOOL;		(*Выход на включение первого насоса.*)
	pump2ON: BOOL;		(*Выход на включение второго насоса.*)
	rTrigPump1ON: R_TRIG;		(*Детектор переднего фронта на запуск насоса 1.*)
	rTrigPump2ON: R_TRIG;		(*Детектор переднего фрона на запуск насоса 2.*)
	rTrigKM1off: R_TRIG;		(*Детектор переднего фронта сигнала на запуск одного из насосов,
			для выключения контактора КМ1 питающего ЧРП.*)
	rsTrigKM1: RS;		(*Триггер управления КМ1 (питание ЧРП).*)
	rsTrigKMpump1: RS;		(*Триггер контактора насоса 1.*)
	rsTrigKMpump2: RS;		(*Триггер контактора насоса 2.*)
	timerKM1off: TOF;		(*Таймер выключения контактора питания ЧРП.*)
	timerKM2DelayON: TON;		(*Таймер задержки включения контактора насоса 1.*)
	timerKM3DelayON: TON;		(*Таймер задержки включения контактора насоса 2.*)
	timerKM2DelayOFF: TOF;		(*Таймер задержки выключения контактора насоса 1.*)
	timerKM3DelayOFF: TOF;		(*Таймер задержки выключения контактора насоса 2.*)
	timerReadyToStartON: TON;		(*Таймер задержки подачи сигнала о готовности к старту (запуск ЧРП).*)
END_VAR
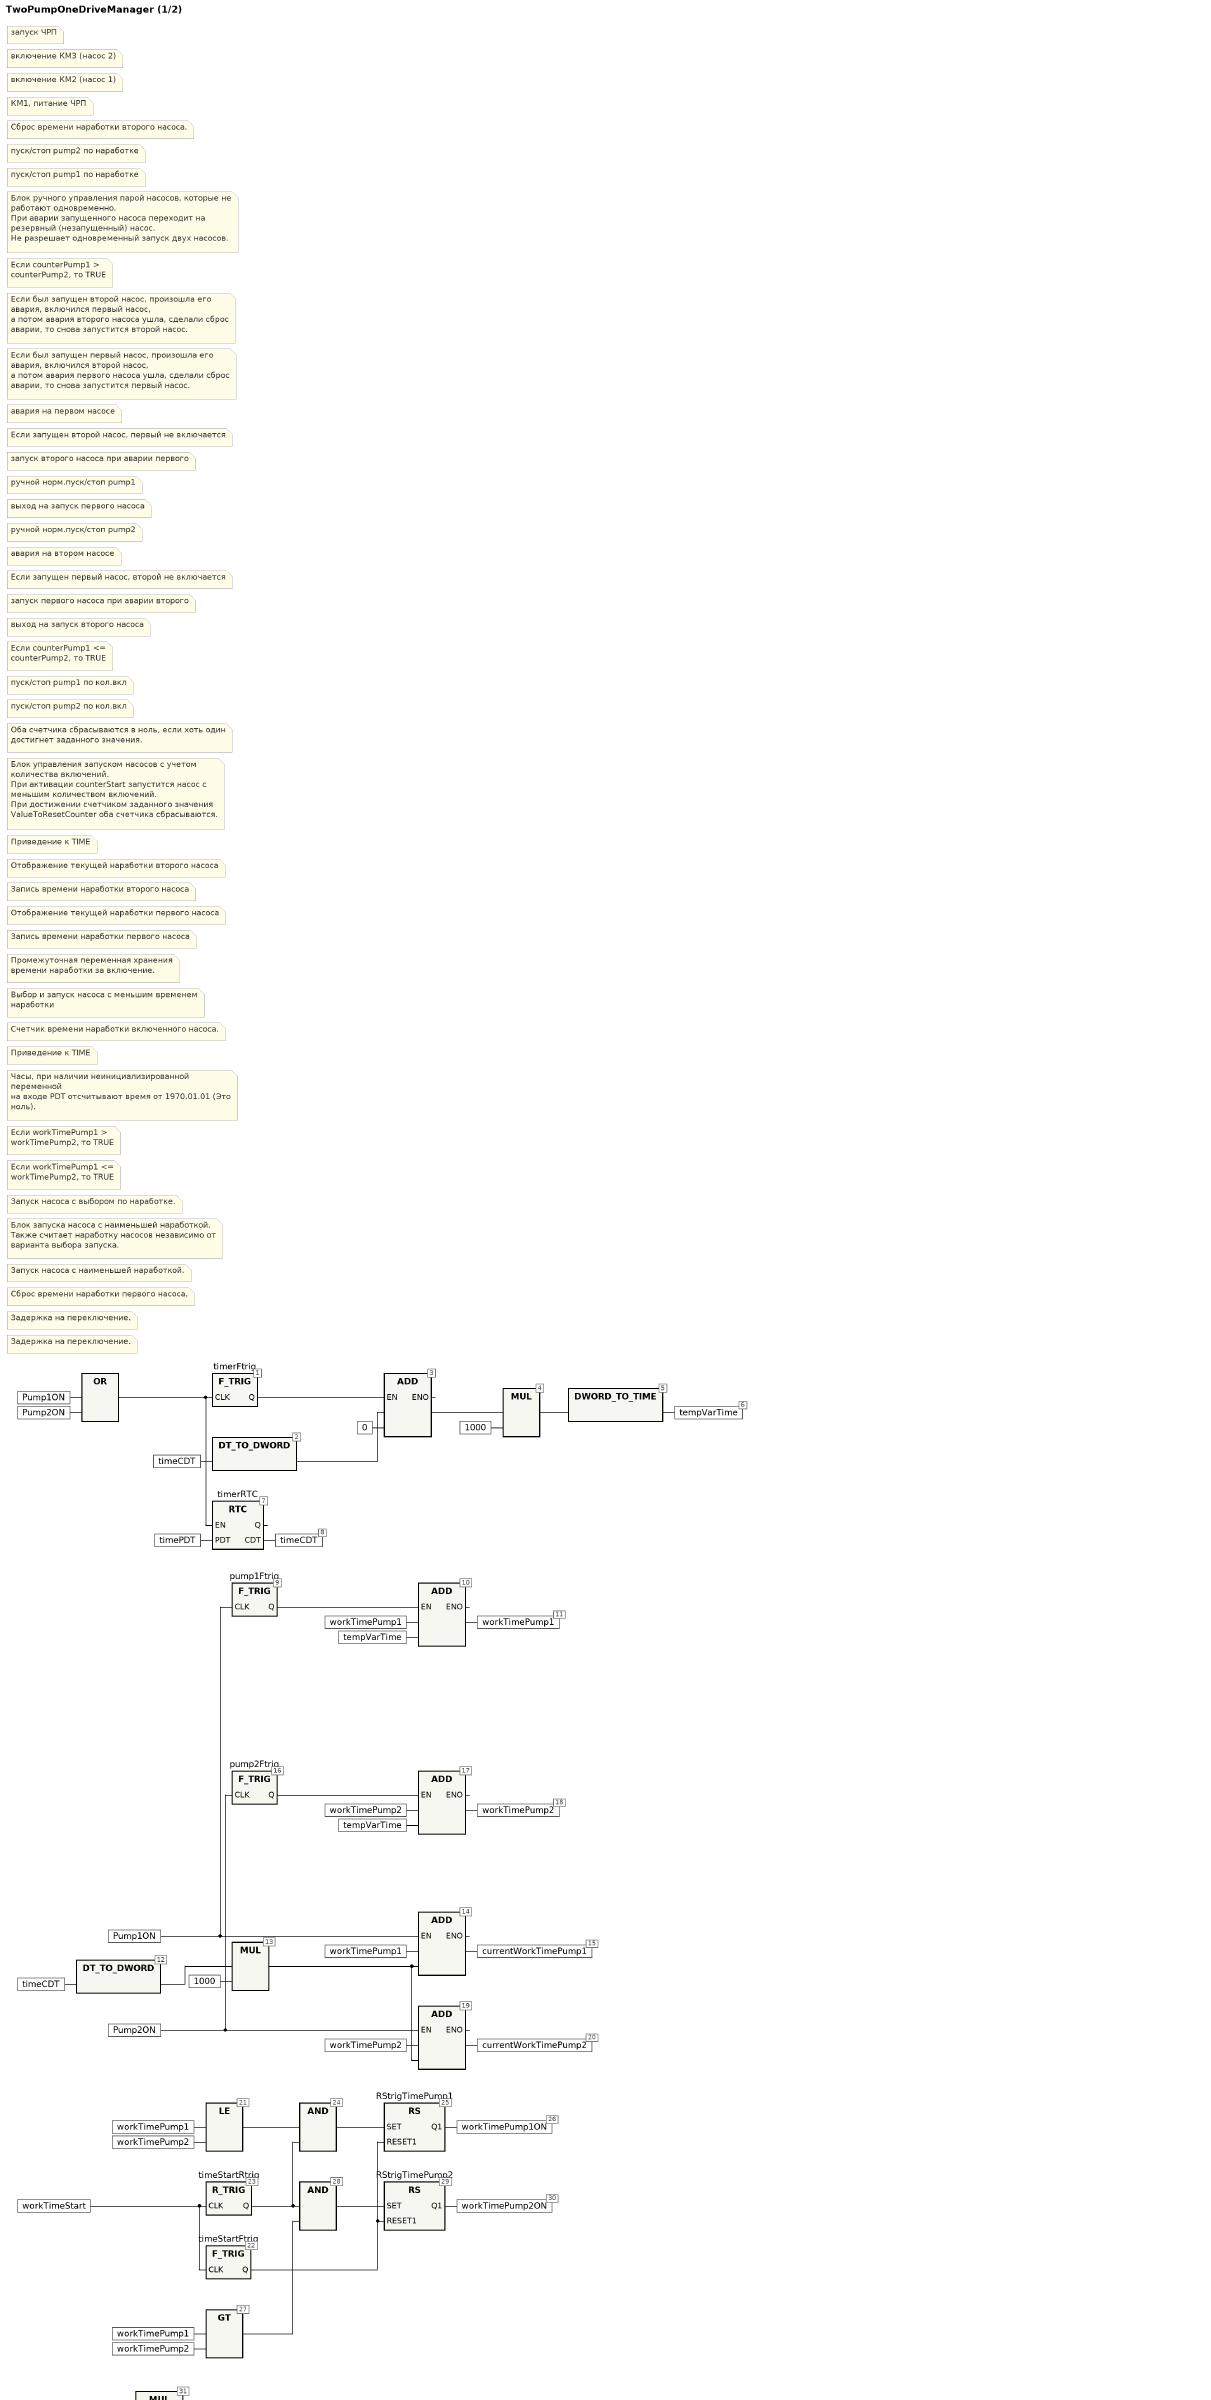
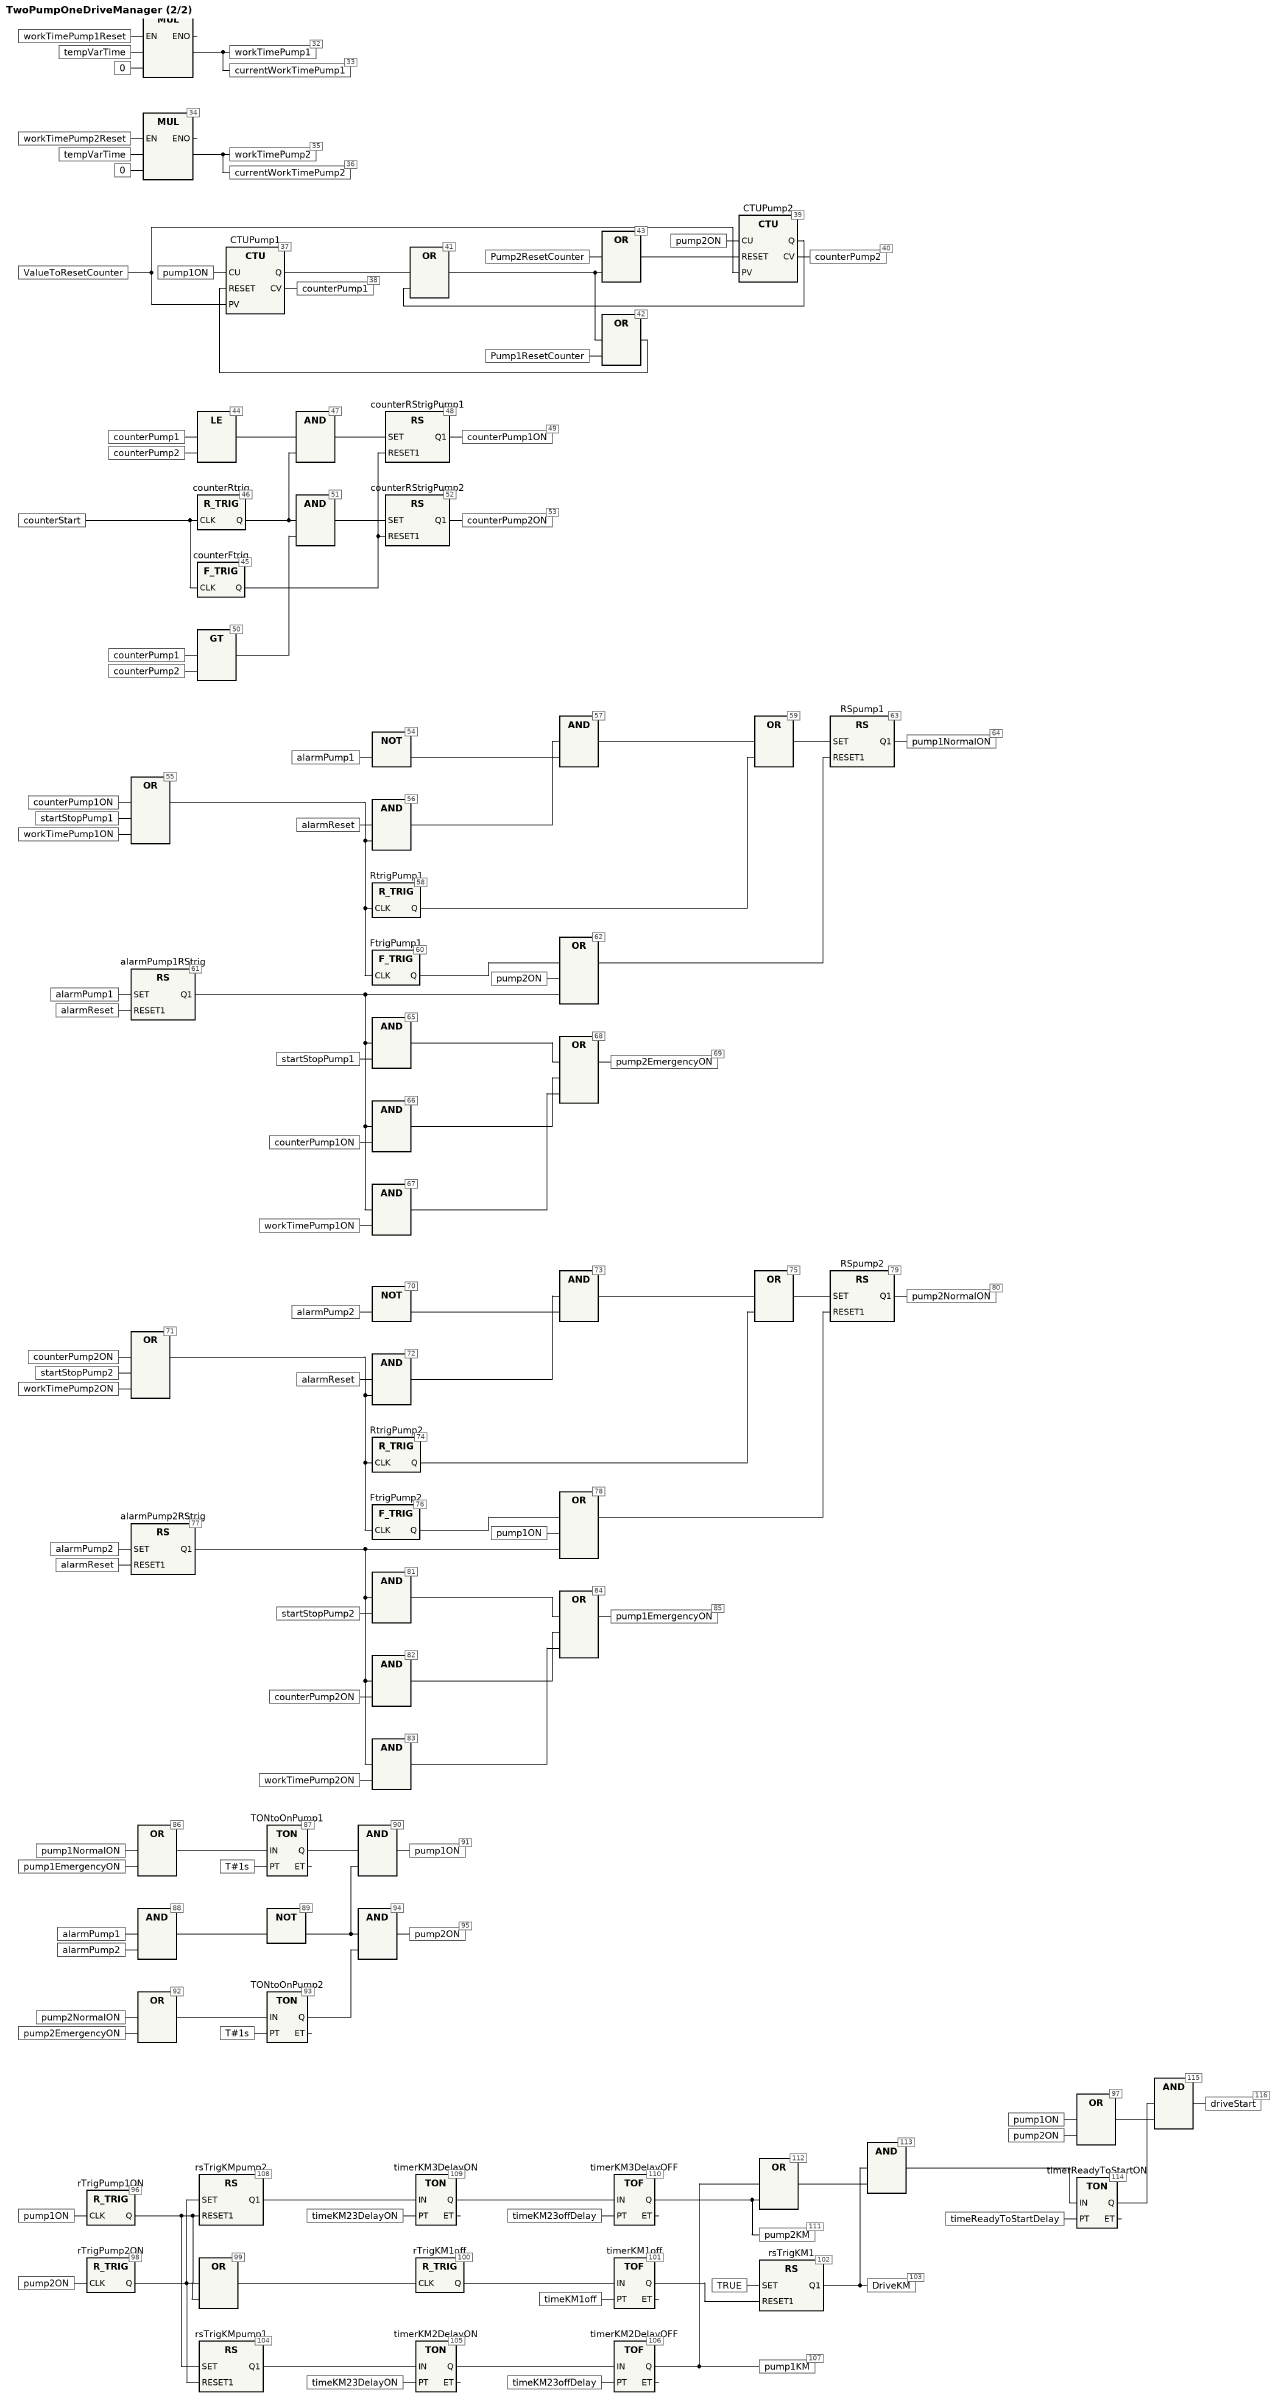
_CFC_ (* Continuous Function Chart, elements in execution order *)
(* запуск ЧРП *)
(* включение КМ3 (насос 2) *)
(* включение КМ2 (насос 1) *)
(* КМ1, питание ЧРП *)
(* Сброс времени наработки второго насоса. *)
(* пуск/стоп pump2 по наработке *)
(* пуск/стоп pump1 по наработке *)
(* Блок ручного управления парой насосов, которые не работают одновременно. / При аварии запущенного насоса переходит на резервный (незапущенный) насос. / Не разрешает одновременный запуск двух насосов. *)
(* Если counterPump1 > / counterPump2, то TRUE *)
(* Если был запущен второй насос, произошла его авария, включился первый насос, / а потом авария второго насоса ушла, сделали сброс аварии, то снова запустится второй насос. *)
(* Если был запущен первый насос, произошла его авария, включился второй насос, / а потом авария первого насоса ушла, сделали сброс аварии, то снова запустится первый насос. *)
(* авария на первом насосе *)
(* Если запущен второй насос, первый не включается *)
(* запуск второго насоса при аварии первого *)
(* ручной норм.пуск/стоп pump1 *)
(* выход на запуск первого насоса *)
(* ручной норм.пуск/стоп pump2 *)
(* авария на втором насосе *)
(* Если запущен первый насос, второй не включается *)
(* запуск первого насоса при аварии второго *)
(* выход на запуск второго насоса *)
(* Если counterPump1 <= / counterPump2, то TRUE *)
(* пуск/стоп pump1 по кол.вкл *)
(* пуск/стоп pump2 по кол.вкл *)
(* Оба счетчика сбрасываются в ноль, если хоть один достигнет заданного значения. *)
(* Блок управления запуском насосов с учетом количества включений. / При активации counterStart запустится насос с меньшим количеством включений. / При достижении счетчиком заданного значения ValueToResetCounter оба счетчика сбрасываются. *)
(* Приведение к TIME *)
(* Отображение текущей наработки второго насоса *)
(* Запись времени наработки второго насоса *)
(* Отображение текущей наработки первого насоса *)
(* Запись времени наработки первого насоса *)
(* Промежуточная переменная хранения / времени наработки за включение. *)
(* Выбор и запуск насоса с меньшим временем наработки *)
(* Счетчик времени наработки включенного насоса. *)
(* Приведение к TIME *)
(* Часы, при наличии неинициализированной переменной / на входе PDT отсчитывают время от 1970.01.01 (Это ноль). *)
(* Если workTimePump1 > / workTimePump2, то TRUE *)
(* Если workTimePump1 <= / workTimePump2, то TRUE *)
(* Запуск насоса с выбором по наработке. *)
(* Блок запуска насоса с наименьшей наработкой. / Также считает наработку насосов независимо от варианта выбора запуска. *)
(* Запуск насоса с наименьшей наработкой. *)
(* Сброс времени наработки первого насоса. *)
(* Задержка на переключение. *)
(* Задержка на переключение. *)
#0 OR(Pump1ON, Pump2ON)
#1 timerFtrig:F_TRIG(CLK: #0)
#2 DT_TO_DWORD(timeCDT)
#3 ADD(EN: #1.Q, #2, 0)
#4 MUL(#3, 1000)
#5 DWORD_TO_TIME(#4)
#6 tempVarTime <= #5
#7 timerRTC:RTC(EN: #0, PDT: timePDT)
#8 timeCDT <= #7.CDT
#9 pump1Ftrig:F_TRIG(CLK: Pump1ON)
#10 ADD(EN: #9.Q, workTimePump1, tempVarTime)
#11 workTimePump1 <= #10
#12 DT_TO_DWORD(timeCDT)
#13 MUL(#12, 1000)
#14 ADD(EN: Pump1ON, workTimePump1, #13)
#15 currentWorkTimePump1 <= #14
#16 pump2Ftrig:F_TRIG(CLK: Pump2ON)
#17 ADD(EN: #16.Q, workTimePump2, tempVarTime)
#18 workTimePump2 <= #17
#19 ADD(EN: Pump2ON, workTimePump2, #13)
#20 currentWorkTimePump2 <= #19
#21 LE(workTimePump1, workTimePump2)
#22 timeStartFtrig:F_TRIG(CLK: workTimeStart)
#23 timeStartRtrig:R_TRIG(CLK: workTimeStart)
#24 AND(#21, #23.Q)
#25 RStrigTimePump1:RS(SET: #24, RESET1: #22.Q)
#26 workTimePump1ON <= #25.Q1
#27 GT(workTimePump1, workTimePump2)
#28 AND(#23.Q, #27)
#29 RStrigTimePump2:RS(SET: #28, RESET1: #22.Q)
#30 workTimePump2ON <= #29.Q1
#31 MUL(EN: workTimePump1Reset, tempVarTime, 0)
#32 workTimePump1 <= #31
#33 currentWorkTimePump1 <= #31
#34 MUL(EN: workTimePump2Reset, tempVarTime, 0)
#35 workTimePump2 <= #34
#36 currentWorkTimePump2 <= #34
#37 CTUPump1:CTU(CU: pump1ON, RESET: #42, PV: ValueToResetCounter)
#38 counterPump1 <= #37.CV
#39 CTUPump2:CTU(CU: pump2ON, RESET: #43, PV: ValueToResetCounter)
#40 counterPump2 <= #39.CV
#41 OR(#37.Q, #39.Q)
#42 OR(#41, Pump1ResetCounter)
#43 OR(Pump2ResetCounter, #41)
#44 LE(counterPump1, counterPump2)
#45 counterFtrig:F_TRIG(CLK: counterStart)
#46 counterRtrig:R_TRIG(CLK: counterStart)
#47 AND(#44, #46.Q)
#48 counterRStrigPump1:RS(SET: #47, RESET1: #45.Q)
#49 counterPump1ON <= #48.Q1
#50 GT(counterPump1, counterPump2)
#51 AND(#46.Q, #50)
#52 counterRStrigPump2:RS(SET: #51, RESET1: #45.Q)
#53 counterPump2ON <= #52.Q1
#54 NOT(alarmPump1)
#55 OR(counterPump1ON, startStopPump1, workTimePump1ON)
#56 AND(alarmReset, #55)
#57 AND(#56, #54)
#58 RtrigPump1:R_TRIG(CLK: #55)
#59 OR(#57, #58.Q)
#60 FtrigPump1:F_TRIG(CLK: #55)
#61 alarmPump1RStrig:RS(SET: alarmPump1, RESET1: alarmReset)
#62 OR(#60.Q, pump2ON, #61.Q1)
#63 RSpump1:RS(SET: #59, RESET1: #62)
#64 pump1NormalON <= #63.Q1
#65 AND(#61.Q1, startStopPump1)
#66 AND(#61.Q1, counterPump1ON)
#67 AND(#61.Q1, workTimePump1ON)
#68 OR(#65, #66, #67)
#69 pump2EmergencyON <= #68
#70 NOT(alarmPump2)
#71 OR(counterPump2ON, startStopPump2, workTimePump2ON)
#72 AND(alarmReset, #71)
#73 AND(#72, #70)
#74 RtrigPump2:R_TRIG(CLK: #71)
#75 OR(#73, #74.Q)
#76 FtrigPump2:F_TRIG(CLK: #71)
#77 alarmPump2RStrig:RS(SET: alarmPump2, RESET1: alarmReset)
#78 OR(#76.Q, pump1ON, #77.Q1)
#79 RSpump2:RS(SET: #75, RESET1: #78)
#80 pump2NormalON <= #79.Q1
#81 AND(#77.Q1, startStopPump2)
#82 AND(#77.Q1, counterPump2ON)
#83 AND(#77.Q1, workTimePump2ON)
#84 OR(#81, #82, #83)
#85 pump1EmergencyON <= #84
#86 OR(pump1NormalON, pump1EmergencyON)
#87 TONtoOnPump1:TON(IN: #86, PT: T#1s)
#88 AND(alarmPump1, alarmPump2)
#89 NOT(#88)
#90 AND(#87.Q, #89)
#91 pump1ON <= #90
#92 OR(pump2NormalON, pump2EmergencyON)
#93 TONtoOnPump2:TON(IN: #92, PT: T#1s)
#94 AND(#89, #93.Q)
#95 pump2ON <= #94
#96 rTrigPump1ON:R_TRIG(CLK: pump1ON)
#97 OR(pump1ON, pump2ON)
#98 rTrigPump2ON:R_TRIG(CLK: pump2ON)
#99 OR(#96.Q, #98.Q)
#100 rTrigKM1off:R_TRIG(CLK: #99)
#101 timerKM1off:TOF(IN: #100.Q, PT: timeKM1off)
#102 rsTrigKM1:RS(SET: TRUE, RESET1: #101.Q)
#103 DriveKM <= #102.Q1
#104 rsTrigKMpump1:RS(SET: #96.Q, RESET1: #98.Q)
#105 timerKM2DelayON:TON(IN: #104.Q1, PT: timeKM23DelayON)
#106 timerKM2DelayOFF:TOF(IN: #105.Q, PT: timeKM23offDelay)
#107 pump1KM <= #106.Q
#108 rsTrigKMpump2:RS(SET: #98.Q, RESET1: #96.Q)
#109 timerKM3DelayON:TON(IN: #108.Q1, PT: timeKM23DelayON)
#110 timerKM3DelayOFF:TOF(IN: #109.Q, PT: timeKM23offDelay)
#111 pump2KM <= #110.Q
#112 OR(#106.Q, #110.Q)
#113 AND(#102.Q1, #112)
#114 timerReadyToStartON:TON(IN: #113, PT: timeReadyToStartDelay)
#115 AND(#114.Q, #97)
#116 driveStart <= #115
_END_CFC_
END_FUNCTION_BLOCK

(* POU CounterTwoPumpManager, CFC *)
FUNCTION_BLOCK CounterTwoPumpManager
VAR_INPUT
	startStopPump1: BOOL;		(*Сигнал на пуск/стоп первого насоса.*)
	startStopPump2: BOOL;		(*Сигнал на пуск/стоп второго насоса.*)
	alarmPump1: BOOL;		(*Сигнал "авария" на первом насосе.*)
	alarmPump2: BOOL;		(*Сигнал "авария" на втором насосе.*)
	alarmReset: BOOL;		(*Сброс аварии.*)

	counterStart: BOOL;		(*Запуск насоса с меньшим количеством включений.*)
	Pump1ResetCounter: BOOL;		(*Сброс счетчика количества включений первого насоса. Сбрасывается также автоматически при достижении счетчиком значения ValueToResetCTU.*)
	Pump2ResetCounter: BOOL;		(*Сброс счетчика количества включений второго насоса. Сбрасывается также автоматически при достижении счетчиком значения ValueToResetCTU.*)
	ValueToResetCounter: WORD := 32767;		(*Значение счетчика, после которого он сбрасывается на ноль.
			Максимальное допустимое значение: 32767, будет установлено, если не подключать ничего на вход.*)
END_VAR
VAR_OUTPUT
	pump1ON: BOOL;		(*Выход на включение первого насоса.*)
	pump2ON: BOOL;		(*Выход на включение второго насоса.*)

	counterPump1: WORD;		(*Количество включений первого насоса. При достижении значения ValueToResetCTU сбрасывается в ноль.*)
	counterPump2: WORD;		(*Количество включений второго насоса. При достижении значения ValueToResetCTU сбрасывается в ноль.*)
END_VAR
VAR
	RtrigPump1: R_TRIG;		(*Включает первый насос по фронту сигнала на ручной пуск/стоп.*)
	FtrigPump1: F_TRIG;		(*Выключает первый насос по спаду сигнала на ручной пуск/стоп.*)
	RtrigPump2: R_TRIG;		(*Включает второй насос по фронту сигнала на ручной пуск/стоп.*)
	FtrigPump2: F_TRIG;		(*Выключает второй насос по спаду сигнала на ручной пуск/стоп.*)
	RSpump1: RS;		(*RS-триггер нормального включения первого насоса*)
	RSpump2: RS;		(*RS-триггер нормального включения второго насоса*)
	pump1NormalON: BOOL;		(*Сигнал нормального (неаварийного) включения первого насоса.*)
	pump2NormalON: BOOL;		(*Сигнал нормального (неаварийного) включения второго насоса.*)
	pump2EmergencyON: BOOL;		(*Сигнал аварийного включения второго насоса (при аварии первого).*)
	pump1EmergencyON: BOOL;		(*Сигнал аварийного включения первого насоса (при аварии второго).*)
	alarmPump1RStrig: RS;		(*Триггер аварии первого насоса.*)
	alarmPump2RStrig: RS;		(*Триггер аварии второго насоса.*)
	TONtoOnPump1: TON;		(*Таймер задержки включения первого насоса, на переключение контакторов при аварийном переключении.
			Жестко задано 1 секунда.*)
	TONtoOnPump2: TON;		(*Таймер задержки включения второго насоса, на переключение контакторов при аварийном переключении.
						Жестко задано 1 секунда.*)

